# B&R Automation Studio project ControlPLC_DataDistribution (part 3)

#### Cyclic.sfc
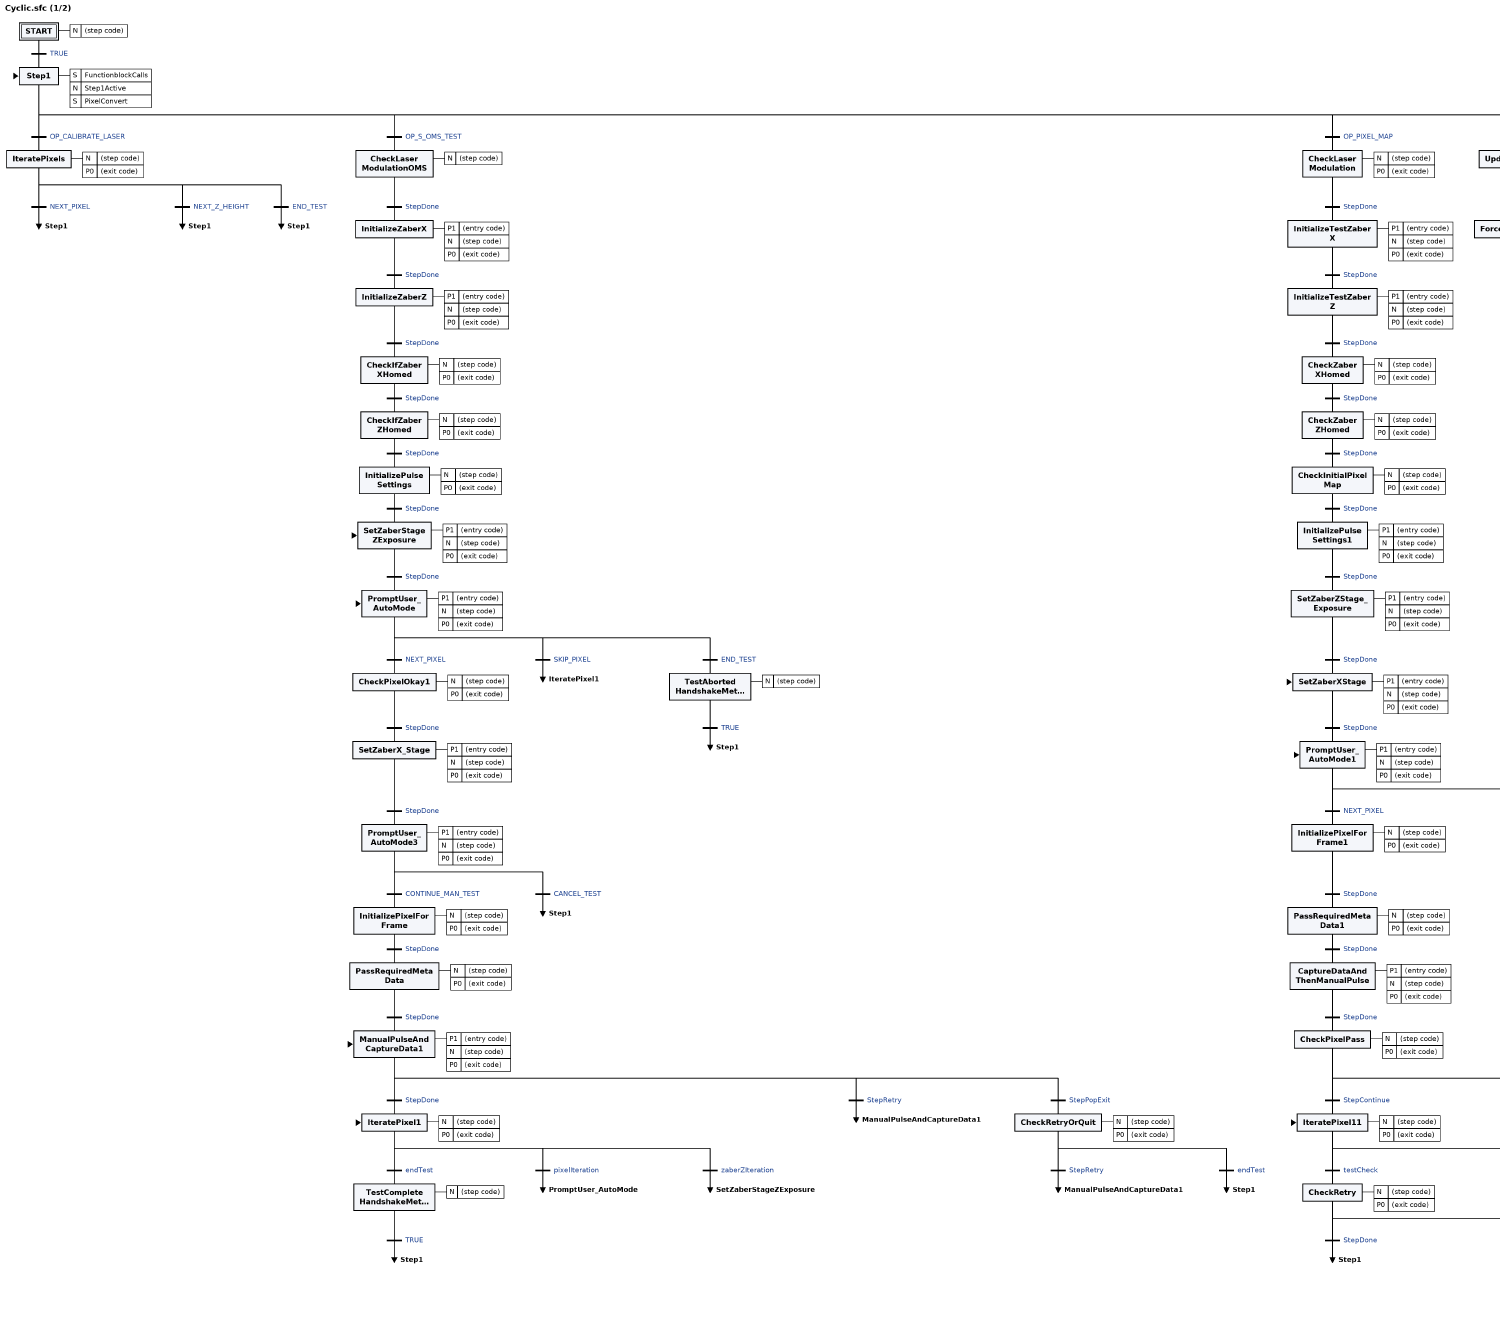
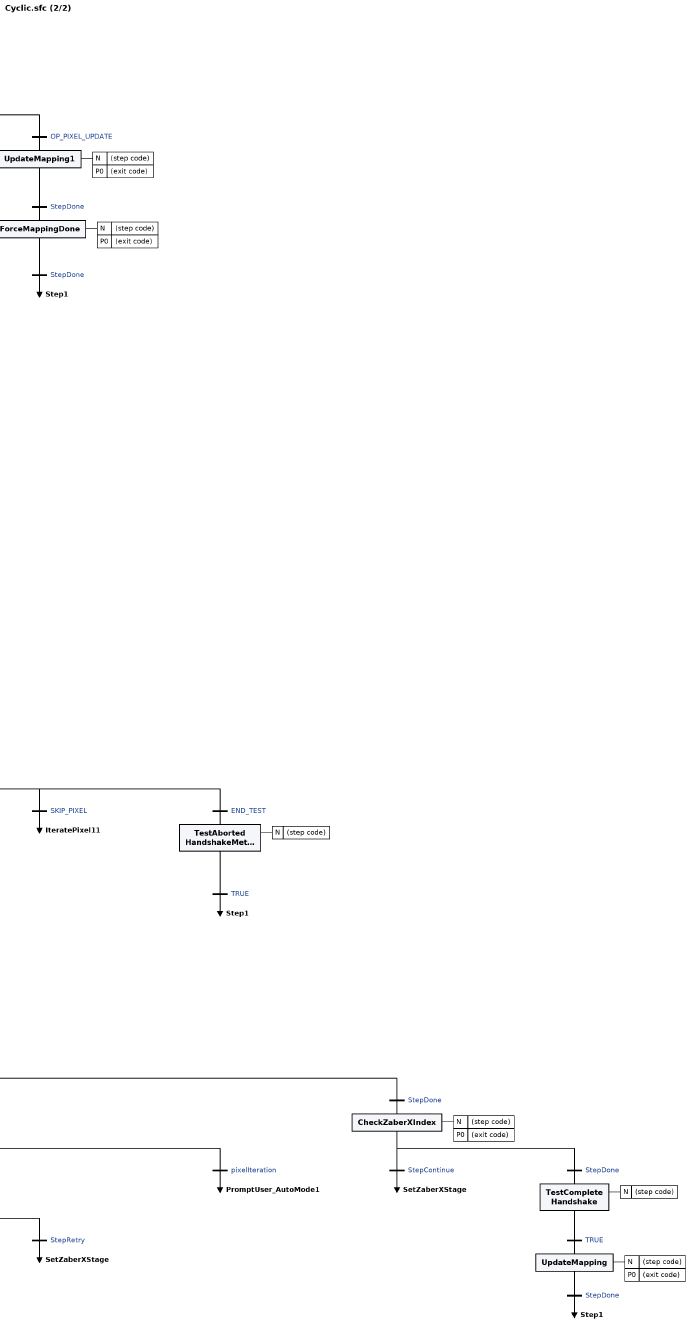
```iecst
PROGRAM _CYCLIC
INITIAL_STEP START:

SFCReset := FALSE;
END_STEP
TRANSITION FROM START TO Step1:=
TRUE
END_TRANSITION
IEC_STEP Step1:
FunctionblockCalls(S);
Step1Active(N);
PixelConvert(S);
END_STEP
TRANSITION FROM Step1 TO IteratePixels:=
OP_CALIBRATE_LASER
END_TRANSITION
TRANSITION FROM Step1 TO CheckLaserModulationOMS:=
OP_S_OMS_TEST
END_TRANSITION
STEP CheckLaserModulationOMS:
OP_S_OMS_TEST := FALSE;
task.internal.activeZaber2Index := 0;

StepDone := TRUE;
END_STEP
TRANSITION FROM CheckLaserModulationOMS TO InitializeZaberX:=
StepDone
END_TRANSITION
STEP InitializeZaberX:
OP_CALIBRATE_LASER := FALSE;
// initialize test
// init meta writer; Zome Zaber

Command.Command := gVFLCR.command.initializeOmsTestZaber1;

Command.Execute := TRUE;
Command();

IF Command.Done THEN
	StepDone := TRUE;
	Command.Execute := FALSE;
	Command();

ELSE
	StepDone := FALSE;
END_IF
END_STEP
ENTRY_ACTION
task.internal.activeZaber2Index := 0;
END_ACTION
EXIT_ACTION
StepDone := FALSE;
(* TODO: Insert Program *)
END_ACTION
TRANSITION FROM InitializeZaberX TO InitializeZaberZ:=
StepDone
END_TRANSITION
STEP InitializeZaberZ:
OP_CALIBRATE_LASER := FALSE;
// initialize test
// init meta writer; Zome Zaber

Command.Command := gVFLCR.command.initializeOmsTestZaber2;

Command.Execute := TRUE;
Command();

IF Command.Done THEN
	StepDone := TRUE;
	Command.Execute := FALSE;
	Command();

ELSE
	StepDone := FALSE;
END_IF
END_STEP
ENTRY_ACTION
task.internal.activeZaber2Index := 0;
END_ACTION
EXIT_ACTION
StepDone := FALSE;
(* TODO: Insert Program *)
END_ACTION
TRANSITION FROM InitializeZaberZ TO CheckIfZaberXHomed:=
StepDone
END_TRANSITION
STEP CheckIfZaberXHomed:
Command.Command := gVFLCR.command.checkZaber1Homed;

Command.Execute := TRUE;
Command();

IF Command.Done THEN
	StepDone := TRUE;
	Command.Execute := FALSE;
	Command();
ELSE
	StepDone := FALSE;
END_IF
END_STEP
EXIT_ACTION
StepDone := FALSE;
(* TODO: Insert Program *)
END_ACTION
TRANSITION FROM CheckIfZaberXHomed TO CheckIfZaberZHomed:=
StepDone
END_TRANSITION
STEP CheckIfZaberZHomed:
Command.Command := gVFLCR.command.checkZaber2Homed;

Command.Execute := TRUE;
Command();

IF Command.Done THEN
	StepDone := TRUE;
	Command.Execute := FALSE;
	Command();
ELSE
	StepDone := FALSE;
END_IF
END_STEP
EXIT_ACTION
StepDone := FALSE;
(* TODO: Insert Program *)
END_ACTION
TRANSITION FROM CheckIfZaberZHomed TO InitializePulseSettings:=
StepDone
END_TRANSITION
STEP InitializePulseSettings:
// initialize app with manual pulse pars; Will create directories for calibration test as well- Should be ok; Assuming data backup of last test to Nas is done by then
Command.Command := gVFLCR.command.initializeCalibration;

Command.pParameters := ADR(gManualPulseTypeSelected);
Command.sParameters := SIZEOF(gManualPulseTypeSelected);

Command.Execute := TRUE;
Command();

IF Command.Done THEN
	StepDone := TRUE;
	Command.Execute := FALSE;
	Command();
ELSE

	StepDone := FALSE;

END_IF
END_STEP
EXIT_ACTION
StepDone := FALSE;
(* TODO: Insert Program *)
END_ACTION
TRANSITION FROM InitializePulseSettings TO SetZaberStageZExposure:=
StepDone
END_TRANSITION
STEP SetZaberStageZExposure:

// Set Zaber height and camera exposure
Command.Command := gVFLCR.command.setZaber2PosAndExposure;

Command.pParameters := ADR(task.internal.adjustZaber2AndCamera);
Command.sParameters := SIZEOF(task.internal.adjustZaber2AndCamera);

Command.Execute := TRUE;
Command();

IF Command.Done THEN
	StepDone := TRUE;
	Command.Execute := FALSE;
	Command();
ELSE

	StepDone := FALSE;

END_IF
END_STEP
ENTRY_ACTION
task.internal.activePixelIndex := 0;

brsmemset( ADR(task.internal.adjustZaber2AndCamera), 0, SIZEOF(task.internal.adjustZaber2AndCamera) );

task.internal.adjustZaber2AndCamera.ZaberAbsolutePos_mm := Configuration.zaber2HeightArray[task.internal.activeZaber2Index];
task.internal.adjustZaber2AndCamera.ZaberMoveAbsolute := TRUE ;
task.internal.adjustZaber2AndCamera.CameraExposure := Configuration.zaber2HeightCameraExpoArray[task.internal.activeZaber2Index];
END_ACTION
EXIT_ACTION
StepDone := FALSE;
END_ACTION
TRANSITION FROM SetZaberStageZExposure TO PromptUser_AutoMode:=
StepDone
END_TRANSITION
STEP PromptUser_AutoMode:

IF NOT autoMode THEN

	task.internal.showPopUp := TRUE;
	task.internal.showNextPixel := TRUE;
	task.internal.showSkipPixel:= TRUE;

	IF task.internal.showPopUp THEN

		IF task.internal.activePixelIndex >= MACHINE_NUM_LASERS_TOTAL THEN

			task.internal.showNextPixel := FALSE;
			task.internal.showSkipPixel:= FALSE;

		ELSIF gVFLCR.status.vfpMap[task.internal.activePixelIndex , 1] = FALSE THEN

			// pixel is disabled
			//task.internal.msgId := TRUE;
			task.internal.showNextPixel := FALSE;

		ELSE

			// pixel is enabled
			//task.internal.msgId := TRUE;
			task.internal.showSkipPixel:= FALSE;

		END_IF

	END_IF

	IF task.internal.showPopUp <> 0 THEN

	END_IF

	//	IF messageHandler.cancel THEN
	//		messageHandler.cancel := 0;
	//		task.internal.msgId := FALSE;
	//		SFCReset := TRUE;
	//		gMachine.IN.CMD.Stop:= TRUE;
	//	END_IF

	//Once a selection is made we are good
	IF NEXT_PIXEL OR SKIP_PIXEL OR END_TEST THEN

		task.internal.showPopUp := FALSE;
		task.internal.showSkipPixel:= FALSE;
		task.internal.showNextPixel := FALSE;

	END_IF
ELSE
	IF gVFLCR.status.vfpMap[task.internal.activePixelIndex, 1] = FALSE THEN
		SKIP_PIXEL := TRUE;
	ELSE
		NEXT_PIXEL := TRUE;
	END_IF
END_IF
END_STEP
ENTRY_ACTION
task.internal.showPopUp := 0;
NEXT_PIXEL := FALSE;
SKIP_PIXEL := FALSE;
END_TEST := FALSE;

END_ACTION
EXIT_ACTION
NEXT_PIXEL := FALSE;
SKIP_PIXEL := FALSE;
END_TEST := FALSE;
END_ACTION
TRANSITION FROM PromptUser_AutoMode TO CheckPixelOkay1:=
NEXT_PIXEL
END_TRANSITION
TRANSITION FROM PromptUser_AutoMode TO IteratePixel1:=
SKIP_PIXEL
END_TRANSITION
(* @SFCISJUMP := 'IteratePixel1' *)
TRANSITION FROM PromptUser_AutoMode TO TestAbortedHandshakeMetaWriter:=
END_TEST
END_TRANSITION
STEP TestAbortedHandshakeMetaWriter:
Command.Command := gVFLCR.command.passAbortedHandshake;

Command.Execute := TRUE;
Command();

IF Command.Done THEN
	StepDone := TRUE;
	Command.Execute := FALSE;
	Command();
ELSE
	StepDone := FALSE;
END_IF
END_STEP
TRANSITION FROM TestAbortedHandshakeMetaWriter TO Step1:=
TRUE
END_TRANSITION
(* @SFCISJUMP := 'Step1' *)
STEP CheckPixelOkay1:
Command.Command := gVFLCR.command.checkMotionOk;
Command.Execute := TRUE;
Command();

IF Command.Done THEN
	StepDone := TRUE;
	Command.Execute := FALSE;
	Command();
ELSE
	StepDone := FALSE;
END_IF

END_STEP
EXIT_ACTION
StepDone := FALSE;
END_ACTION
TRANSITION FROM CheckPixelOkay1 TO SetZaberX_Stage:=
StepDone
END_TRANSITION
STEP SetZaberX_Stage:

// Set Zaber height and camera exposure
Command.Command := gVFLCR.command.setZaber1Pos;

Command.pParameters := ADR(task.internal.adjustZaber1);
Command.sParameters := SIZEOF(task.internal.adjustZaber1);

Command.Execute := TRUE;
Command();

IF Command.Done THEN
	StepDone := TRUE;
	Command.Execute := FALSE;
	Command();
ELSE

	StepDone := FALSE;

END_IF
END_STEP
ENTRY_ACTION

brsmemset( ADR(task.internal.adjustZaber1), 0, SIZEOF(task.internal.adjustZaber1) );

task.internal.adjustZaber1.ZaberAbsolutePos_mm := Configuration.zaber1Position + ((task.internal.activePixelIndex+1) * OPTICS_BOX_PIXEL_XY_OFFSET) ;
task.internal.adjustZaber1.ZaberMoveAbsolute := TRUE ;

END_ACTION
EXIT_ACTION
StepDone := FALSE;
END_ACTION
TRANSITION FROM SetZaberX_Stage TO PromptUser_AutoMode3:=
StepDone
END_TRANSITION
STEP PromptUser_AutoMode3:

IF NOT autoMode THEN

	task.internal.pausePopUp := TRUE;
	task.internal.continuePopUp := TRUE;
	task.internal.cancelPopUp := TRUE;

	IF task.internal.pausePopUp <> 0 THEN

	END_IF

	//Once a selection is made we are good
	IF CONTINUE_MAN_TEST OR CANCEL_TEST THEN

		task.internal.pausePopUp := FALSE;
		task.internal.continuePopUp:= FALSE;
		task.internal.cancelPopUp := FALSE;

	END_IF
ELSE
	CONTINUE_MAN_TEST := TRUE;
	task.internal.pausePopUp := FALSE;
	task.internal.continuePopUp:= FALSE;
	task.internal.cancelPopUp := FALSE;
END_IF
END_STEP
ENTRY_ACTION
task.internal.pausePopUp := 0;
CONTINUE_MAN_TEST := FALSE;
CANCEL_TEST := FALSE;

END_ACTION
EXIT_ACTION
CONTINUE_MAN_TEST := FALSE;
CANCEL_TEST := FALSE;
END_ACTION
TRANSITION FROM PromptUser_AutoMode3 TO InitializePixelForFrame:=
CONTINUE_MAN_TEST
END_TRANSITION
TRANSITION FROM PromptUser_AutoMode3 TO Step1:=
CANCEL_TEST
END_TRANSITION
(* @SFCISJUMP := 'Step1' *)
STEP InitializePixelForFrame:
Command.Command := gVFLCR.command.initializePixelForFrame;

task.internal.initializePixelParameters.activePixelIndex := task.internal.activePixelIndex;

Command.pParameters := ADR(task.internal.initializePixelParameters);
Command.sParameters := SIZEOF(task.internal.initializePixelParameters);

Command.Execute := TRUE;
Command();

IF Command.Done THEN
	StepDone := TRUE;
	Command.Execute := FALSE;
	Command();
ELSE

	StepDone := FALSE;

END_IF
END_STEP
EXIT_ACTION
StepDone := FALSE;
END_ACTION
TRANSITION FROM InitializePixelForFrame TO PassRequiredMetaData:=
StepDone
END_TRANSITION
STEP PassRequiredMetaData:
Command.Command := gVFLCR.command.passRequiredMetaData;

Command.Execute := TRUE;
Command();

IF Command.Done THEN
	StepDone := TRUE;
	Command.Execute := FALSE;
	Command();
ELSE
	StepDone := FALSE;
END_IF
END_STEP
EXIT_ACTION
StepDone := FALSE;
END_ACTION
TRANSITION FROM PassRequiredMetaData TO ManualPulseAndCaptureData1:=
StepDone
END_TRANSITION
STEP ManualPulseAndCaptureData1:
Command.Command := gVFLCR.command.manualPulse;

Command.pParameters := ADR(task.internal.manualPulse);
Command.sParameters := SIZEOF(task.internal.manualPulse);

Command.Execute := TRUE;
Command();

IF Command.Done THEN
	StepDone := TRUE;
	task.internal.failedImageCaptureRetry := 0;
	Command.Execute := FALSE;
	Command();
ELSIF Command.Error THEN
	IF task.internal.failedImageCaptureRetry < task.internal.numOfRetries THEN
		StepRetry := TRUE;
		task.internal.failedImageCaptureRetry := task.internal.failedImageCaptureRetry +1;
		Command.Execute := FALSE;
		Command();
	ELSE
		task.internal.failedImageCaptureRetry := 0;
		StepDone := FALSE;
		StepRetry := FALSE;
		StepPopExit := TRUE;
		Command.Execute := FALSE;
		Command();
	END_IF
ELSE
	StepDone := FALSE;
END_IF
END_STEP
ENTRY_ACTION
task.internal.numOfRetries := 4;
END_ACTION
EXIT_ACTION
StepRetry := FALSE;
StepDone := FALSE;
StepPopExit := FALSE;
END_ACTION
TRANSITION FROM ManualPulseAndCaptureData1 TO IteratePixel1:=
StepDone
END_TRANSITION
TRANSITION FROM ManualPulseAndCaptureData1 TO ManualPulseAndCaptureData1:=
StepRetry
END_TRANSITION
(* @SFCISJUMP := 'ManualPulseAndCaptureData1' *)
TRANSITION FROM ManualPulseAndCaptureData1 TO CheckRetryOrQuit:=
StepPopExit
END_TRANSITION
STEP CheckRetryOrQuit:
task.internal.showErrorMessage := TRUE;

IF task.internal.showErrorMessage <> 0 THEN

END_IF

IF CLOSE_POPUP  THEN

	task.internal.showErrorMessage := FALSE;
	endTest :=TRUE;
	StepRetry:=FALSE;

END_IF

IF RETRY_POPUP  THEN

	task.internal.showErrorMessage := FALSE;
	StepRetry:=TRUE;
	endTest :=FALSE;

END_IF
END_STEP
EXIT_ACTION
endTest := FALSE;
StepRetry := FALSE;
END_ACTION
TRANSITION FROM CheckRetryOrQuit TO ManualPulseAndCaptureData1:=
StepRetry
END_TRANSITION
(* @SFCISJUMP := 'ManualPulseAndCaptureData1' *)
TRANSITION FROM CheckRetryOrQuit TO Step1:=
endTest
END_TRANSITION
(* @SFCISJUMP := 'Step1' *)
STEP IteratePixel1:
task.internal.activePixelIndex := task.internal.activePixelIndex + 1;

IF task.internal.activePixelIndex >= MACHINE_NUM_LASERS_TOTAL THEN
	IF  task.internal.activeZaber2Index < 10 THEN // 0-10 point reading with 5 being zero offset position and 5 reading on either side
		zaberZIteration := TRUE;
		task.internal.activeZaber2Index := task.internal.activeZaber2Index + 1;
	ELSE
		endTest := TRUE;
	END_IF
ELSE
	pixelIteration := TRUE;
END_IF
END_STEP
EXIT_ACTION

pixelIteration := FALSE;
zaberZIteration := FALSE;
endTest := FALSE;
END_ACTION
TRANSITION FROM IteratePixel1 TO TestCompleteHandshakeMetaWriter:=
endTest
END_TRANSITION
TRANSITION FROM IteratePixel1 TO PromptUser_AutoMode:=
pixelIteration
END_TRANSITION
(* @SFCISJUMP := 'PromptUser_AutoMode' *)
TRANSITION FROM IteratePixel1 TO SetZaberStageZExposure:=
zaberZIteration
END_TRANSITION
(* @SFCISJUMP := 'SetZaberStageZExposure' *)
STEP TestCompleteHandshakeMetaWriter:
endTest := FALSE;

Command.Command := gVFLCR.command.passCompleteHandshake;

Command.Execute := TRUE;
Command();

IF Command.Done THEN
	StepDone := TRUE;
	omsTestComplete := TRUE;
	Command.Execute := FALSE;
	Command();
ELSE
	StepDone := FALSE;
END_IF
END_STEP
TRANSITION FROM TestCompleteHandshakeMetaWriter TO Step1:=
TRUE
END_TRANSITION
(* @SFCISJUMP := 'Step1' *)
TRANSITION FROM Step1 TO CheckLaserModulation:=
OP_PIXEL_MAP
END_TRANSITION
STEP CheckLaserModulation:
OP_PIXEL_MAP := FALSE;
omsTestComplete := FALSE;
endTest := FALSE;
pixelIteration := FALSE;

FOR loopVar := 0 TO MACHINE_MAI_LASERS_TOTAL BY 1 DO
	pixelIgnoreList[loopVar] := FALSE;
END_FOR

StepDone := TRUE;

END_STEP
EXIT_ACTION
StepDone := FALSE;
END_ACTION
TRANSITION FROM CheckLaserModulation TO InitializeTestZaberX:=
StepDone
END_TRANSITION
STEP InitializeTestZaberX:
OP_CALIBRATE_LASER := FALSE;
// initialize test
// init meta writer; Zome Zaber

Command.Command := gVFLCR.command.initializeOmsTestZaber1;

Command.Execute := TRUE;
Command();

IF Command.Done THEN
	StepDone := TRUE;
	Command.Execute := FALSE;
	Command();

ELSE
	StepDone := FALSE;
END_IF
END_STEP
ENTRY_ACTION
task.internal.activeZaber2Index := 0;
END_ACTION
EXIT_ACTION
StepDone := FALSE;
END_ACTION
TRANSITION FROM InitializeTestZaberX TO InitializeTestZaberZ:=
StepDone
END_TRANSITION
STEP InitializeTestZaberZ:
OP_CALIBRATE_LASER := FALSE;
// initialize test
// init meta writer; Zome Zaber

Command.Command := gVFLCR.command.initializeOmsTestZaber2;

Command.Execute := TRUE;
Command();

IF Command.Done THEN
	StepDone := TRUE;
	Command.Execute := FALSE;
	Command();

ELSE
	StepDone := FALSE;
END_IF
END_STEP
ENTRY_ACTION
task.internal.activeZaber2Index := 0;
END_ACTION
EXIT_ACTION
StepDone := FALSE;
END_ACTION
TRANSITION FROM InitializeTestZaberZ TO CheckZaberXHomed:=
StepDone
END_TRANSITION
STEP CheckZaberXHomed:
Command.Command := gVFLCR.command.checkZaber1Homed;

Command.Execute := TRUE;
Command();

IF Command.Done THEN
	StepDone := TRUE;
	Command.Execute := FALSE;
	Command();
ELSE
	StepDone := FALSE;
END_IF
END_STEP
EXIT_ACTION
StepDone := FALSE;
END_ACTION
TRANSITION FROM CheckZaberXHomed TO CheckZaberZHomed:=
StepDone
END_TRANSITION
STEP CheckZaberZHomed:
Command.Command := gVFLCR.command.checkZaber2Homed;

Command.Execute := TRUE;
Command();

IF Command.Done THEN
	StepDone := TRUE;
	Command.Execute := FALSE;
	Command();
ELSE
	StepDone := FALSE;
END_IF
END_STEP
EXIT_ACTION
StepDone := FALSE;
END_ACTION
TRANSITION FROM CheckZaberZHomed TO CheckInitialPixelMap:=
StepDone
END_TRANSITION
STEP CheckInitialPixelMap:
task.status.allPixelsMapped := stateAllTrue(gVFLCR.status.pixelMapped, FALSE);

FOR task.internal.rackNumber := 0 TO MACHINE_MAI_LASER_RACKS  DO
	FOR task.internal.laserNumber := 0 TO MACHINE_MAI_LASERS_PER_RACK  DO
		gVFLCR.status.vfpMap[task.internal.laserNumber,task.internal.rackNumber] := TRUE;
		//task.internal.laserNumber := task.internal.laserNumber +1;
	END_FOR
	//task.internal.rackNumber := task.internal.rackNumber +1;
END_FOR

IF task.status.allPixelsMapped THEN
	StepDone := TRUE;
ELSE
	StepDone := FALSE;

	Command.Command := gVFLCR.command.laserRackRemap;

	Command.Execute := TRUE;
	Command();

	IF Command.Done THEN
		StepDone := TRUE;
		Command.Execute := FALSE;
		Command();
	ELSIF Command.Error THEN
		StepError := TRUE;
	END_IF

END_IF
END_STEP
EXIT_ACTION
StepDone := FALSE;
END_ACTION
TRANSITION FROM CheckInitialPixelMap TO InitializePulseSettings1:=
StepDone
END_TRANSITION
STEP InitializePulseSettings1:
// initialize app with manual pulse pars; Will create directories for calibration test as well- Should be ok; Assuming data backup of last test to Nas is done by then
Command.Command := gVFLCR.command.initializeCalibration;

Command.pParameters := ADR(gManualPulseTypeSelected);
Command.sParameters := SIZEOF(gManualPulseTypeSelected);

Command.Execute := TRUE;
Command();

IF Command.Done THEN
	StepDone := TRUE;
	Command.Execute := FALSE;
	Command();
ELSE

	StepDone := FALSE;

END_IF
END_STEP
ENTRY_ACTION
brsmemset(ADR(derivedMappingList), 0, SIZEOF(derivedMappingList));
END_ACTION
EXIT_ACTION
StepDone := FALSE;
END_ACTION
TRANSITION FROM InitializePulseSettings1 TO SetZaberZStage_Exposure:=
StepDone
END_TRANSITION
STEP SetZaberZStage_Exposure:

task.internal.adjustZaber1.ZaberAbsolutePos_mm := Configuration.zaber1Position;
// Set Zaber height and camera exposure
Command.Command := gVFLCR.command.setZaber2PosAndExposure;

Command.pParameters := ADR(task.internal.adjustZaber2AndCamera);
Command.sParameters := SIZEOF(task.internal.adjustZaber2AndCamera);

Command.Execute := TRUE;
Command();

IF Command.Done THEN
	StepDone := TRUE;
	Command.Execute := FALSE;
	Command();
ELSE

	StepDone := FALSE;

END_IF
END_STEP
ENTRY_ACTION

task.internal.actualPixelMapIndex :=0; // used for derived mapping list
task.internal.activeZaber1Index := 0; // Initialized once at the start of the test
task.internal.failedImageCaptureRetry := 0; // Reset Retry count

brsmemset( ADR(task.internal.adjustZaber2AndCamera), 0, SIZEOF(task.internal.adjustZaber2AndCamera) );

task.internal.adjustZaber2AndCamera.ZaberAbsolutePos_mm := Configuration.zaber2HeightArray[5]; // only use middle height
task.internal.adjustZaber2AndCamera.ZaberMoveAbsolute := TRUE ;
task.internal.adjustZaber2AndCamera.CameraExposure := Configuration.zaber2HeightCameraExpoArray[5];
END_ACTION
EXIT_ACTION
StepDone := FALSE;
END_ACTION
TRANSITION FROM SetZaberZStage_Exposure TO SetZaberXStage:=
StepDone
END_TRANSITION
STEP SetZaberXStage:

// Set Zaber height and camera exposure
Command.Command := gVFLCR.command.setZaber1Pos;

FOR loopVar := 0 TO MACHINE_MAI_LASERS_TOTAL BY 1 DO
	IF pixelIgnoreList[task.internal.activePixelIndex] = TRUE THEN
		task.internal.activePixelIndex := task.internal.activePixelIndex + 1;
	ELSE
		EXIT;
	END_IF
END_FOR

Command.pParameters := ADR(task.internal.adjustZaber1);
Command.sParameters := SIZEOF(task.internal.adjustZaber1);

Command.Execute := TRUE;
Command();

IF Command.Done THEN
	StepDone := TRUE;
	Command.Execute := FALSE;
	Command();
ELSE

	StepDone := FALSE;

END_IF
END_STEP
ENTRY_ACTION
task.internal.activePixelIndex := 0; // used to iterate through all pixels during pixel mapping

FOR loopVar := 0 TO MACHINE_MAI_LASERS_TOTAL BY 1 DO
	IF pixelIgnoreList[task.internal.activePixelIndex] = TRUE THEN
		task.internal.activePixelIndex := task.internal.activePixelIndex + 1;
	ELSE
		EXIT;
	END_IF
END_FOR

brsmemset( ADR(task.internal.adjustZaber1), 0, SIZEOF(task.internal.adjustZaber1) );

task.internal.adjustZaber1.ZaberAbsolutePos_mm := Configuration.zaber1Position + ((task.internal.activeZaber1Index+1) * OPTICS_BOX_PIXEL_XY_OFFSET) ;
task.internal.adjustZaber1.ZaberMoveAbsolute := TRUE ;

END_ACTION
EXIT_ACTION
StepDone := FALSE;
END_ACTION
TRANSITION FROM SetZaberXStage TO PromptUser_AutoMode1:=
StepDone
END_TRANSITION
STEP PromptUser_AutoMode1:

IF NOT autoMode THEN
	task.internal.showPopUp := TRUE;
	task.internal.showNextPixel := TRUE;
	task.internal.showSkipPixel:= TRUE;

	IF task.internal.showPopUp THEN

		IF task.internal.activePixelIndex >= MACHINE_NUM_LASERS_TOTAL THEN

			task.internal.showNextPixel := FALSE;
			task.internal.showSkipPixel:= FALSE;

		ELSIF pixelIgnoreList[task.internal.activePixelIndex] = TRUE THEN

			// pixel is disabled
			//task.internal.msgId := TRUE;
			task.internal.showNextPixel := FALSE;

		ELSE

			// pixel is enabled
			//task.internal.msgId := TRUE;
			task.internal.showSkipPixel:= FALSE;

		END_IF

	END_IF

	IF task.internal.showPopUp <> 0 THEN

	END_IF

	//	IF messageHandler.cancel THEN
	//		messageHandler.cancel := 0;
	//		task.internal.msgId := FALSE;
	//		SFCReset := TRUE;
	//		gMachine.IN.CMD.Stop:= TRUE;
	//	END_IF

	//Once a selection is made we are good
	IF NEXT_PIXEL OR SKIP_PIXEL OR END_TEST THEN

		task.internal.showPopUp := FALSE;
		task.internal.showSkipPixel:= FALSE;
		task.internal.showNextPixel := FALSE;

	END_IF
ELSE
	IF pixelIgnoreList[task.internal.activePixelIndex] = TRUE THEN
		SKIP_PIXEL := TRUE;
	ELSE
		NEXT_PIXEL := TRUE;
	END_IF
END_IF
END_STEP
ENTRY_ACTION
task.internal.showPopUp := 0;
NEXT_PIXEL := FALSE;
SKIP_PIXEL := FALSE;
END_TEST := FALSE;
END_ACTION
EXIT_ACTION
NEXT_PIXEL := FALSE;
SKIP_PIXEL := FALSE;
END_TEST := FALSE;
END_ACTION
TRANSITION FROM PromptUser_AutoMode1 TO InitializePixelForFrame1:=
NEXT_PIXEL
END_TRANSITION
TRANSITION FROM PromptUser_AutoMode1 TO IteratePixel11:=
SKIP_PIXEL
END_TRANSITION
(* @SFCISJUMP := 'IteratePixel11' *)
TRANSITION FROM PromptUser_AutoMode1 TO TestAbortedHandshakeMetaWriter1:=
END_TEST
END_TRANSITION
STEP TestAbortedHandshakeMetaWriter1:
Command.Command := gVFLCR.command.passAbortedHandshake;

Command.Execute := TRUE;
Command();

IF Command.Done THEN
	StepDone := TRUE;
	Command.Execute := FALSE;
	Command();
ELSE
	StepDone := FALSE;
END_IF
END_STEP
TRANSITION FROM TestAbortedHandshakeMetaWriter1 TO Step1:=
TRUE
END_TRANSITION
(* @SFCISJUMP := 'Step1' *)
STEP InitializePixelForFrame1:
Command.Command := gVFLCR.command.initializePixelForFrame;

task.internal.initializePixelParameters.activePixelIndex := task.internal.activePixelIndex;

Command.pParameters := ADR(task.internal.initializePixelParameters);
Command.sParameters := SIZEOF(task.internal.initializePixelParameters);

Command.Execute := TRUE;
Command();

IF Command.Done THEN
	StepDone := TRUE;
	Command.Execute := FALSE;
	Command();
ELSE

	StepDone := FALSE;

END_IF
END_STEP
EXIT_ACTION
StepDone := FALSE;
END_ACTION
TRANSITION FROM InitializePixelForFrame1 TO PassRequiredMetaData1:=
StepDone
END_TRANSITION
STEP PassRequiredMetaData1:
Command.Command := gVFLCR.command.passRequiredMetaData;

Command.Execute := TRUE;
Command();

IF Command.Done THEN
	StepDone := TRUE;
	Command.Execute := FALSE;
	Command();
ELSE
	StepDone := FALSE;
END_IF
END_STEP
EXIT_ACTION
StepDone := FALSE;
END_ACTION
TRANSITION FROM PassRequiredMetaData1 TO CaptureDataAndThenManualPulse:=
StepDone
END_TRANSITION
STEP CaptureDataAndThenManualPulse:
Command.Command := gVFLCR.command.manualPulse;

Command.pParameters := ADR(task.internal.manualPulse);
Command.sParameters := SIZEOF(task.internal.manualPulse);

Command.Execute := TRUE;
Command();

IF Command.Done THEN
	StepDone := TRUE;
	Command.Execute := FALSE;
	Command();
ELSIF Command.Error THEN
	StepDone := TRUE;
	Command.Execute := FALSE;
	Command();

END_IF
END_STEP
ENTRY_ACTION
task.internal.numOfRetries := 3;
END_ACTION
EXIT_ACTION
StepDone := FALSE;
END_ACTION
TRANSITION FROM CaptureDataAndThenManualPulse TO CheckPixelPass:=
StepDone
END_TRANSITION
STEP CheckPixelPass:
task.internal.rackNumber := 0;
task.internal.laserNumber :=0;

IF gVFLCR.status.frameCaptured THEN
	//task.internal.actualPixelMapIndex := task.internal.actualPixelMapIndex +1;
	FOR task.internal.rackNumber := 0 TO MACHINE_MAI_LASER_RACKS  DO
		IF NOT (gVFLCR.status.vfpMap[task.internal.activePixelIndex, 1] = FALSE) THEN
			FOR task.internal.laserNumber := 0 TO MACHINE_MAI_LASERS_PER_RACK  DO
				IF gmapRackLaser_to_Pixel[task.internal.rackNumber,task.internal.laserNumber] = task.internal.activePixelIndex THEN
					derivedMappingList[task.internal.rackNumber,task.internal.laserNumber] := task.internal.activeZaber1Index;
					pixelIgnoreList[task.internal.activePixelIndex] := TRUE;
					gVFLCR.status.frameCaptured := FALSE;
				END_IF
			END_FOR
		END_IF
	END_FOR
			StepDone := TRUE;
			StepContinue := FALSE;

		ELSE
			StepDone := FALSE;
			StepContinue := TRUE;
		END_IF

END_STEP
EXIT_ACTION
StepDone := FALSE;
StepContinue := FALSE;
END_ACTION
TRANSITION FROM CheckPixelPass TO IteratePixel11:=
StepContinue
END_TRANSITION
TRANSITION FROM CheckPixelPass TO CheckZaberXIndex:=
StepDone
END_TRANSITION
STEP CheckZaberXIndex:
IF task.internal.activeZaber1Index < (MACHINE_NUM_LASERS_TOTAL - 1) THEN
	StepContinue := TRUE;
	task.internal.activeZaber1Index:= task.internal.activeZaber1Index +1 ;
ELSE
	StepDone := TRUE;
END_IF

END_STEP
EXIT_ACTION
StepDone := FALSE;
StepContinue := FALSE;
END_ACTION
TRANSITION FROM CheckZaberXIndex TO SetZaberXStage:=
StepContinue
END_TRANSITION
(* @SFCISJUMP := 'SetZaberXStage' *)
TRANSITION FROM CheckZaberXIndex TO TestCompleteHandshake:=
StepDone
END_TRANSITION
STEP TestCompleteHandshake:
endTest := FALSE;

Command.Command := gVFLCR.command.passCompleteHandshake;

Command.Execute := TRUE;
Command();

IF Command.Done THEN
	StepDone := TRUE;
	omsTestComplete := TRUE;
	Command.Execute := FALSE;
	Command();
ELSE
	StepDone := FALSE;
END_IF
END_STEP
TRANSITION FROM TestCompleteHandshake TO UpdateMapping:=
TRUE
END_TRANSITION
STEP UpdateMapping:

FOR task.internal.rackIndex := 0 TO (MACHINE_NUM_LASER_RACKS-1)  DO
	FOR task.internal.laserIndex := 0 TO (MACHINE_NUM_LASERS_PER_RACK-1) DO

		IF gVFLCR.status.vfpMap[gmapRackLaser_to_Pixel[task.internal.rackIndex,task.internal.laserIndex],1 ] = TRUE
			AND (((task.internal.rackIndex*MACHINE_NUM_LASERS_PER_RACK) + task.internal.laserIndex) < MACHINE_NUM_LASERS_TOTAL) THEN
			gmapRackLaser_to_Pixel[task.internal.rackIndex,task.internal.laserIndex] := derivedMappingList[task.internal.rackIndex,task.internal.laserIndex ];
			//task.internal.laserNumber := task.internal.laserNumber +1;
			gmapPixel_to_Rack[derivedMappingList[task.internal.rackIndex,task.internal.laserIndex]] := task.internal.rackIndex;
			gmapPixel_to_Laser[derivedMappingList[task.internal.rackIndex,task.internal.laserIndex]] := task.internal.laserIndex;
		END_IF
	END_FOR
END_FOR

FOR task.internal.clearListPixelNumber := 0 TO MACHINE_NUM_LASERS_TOTAL-1 DO
	pixelIgnoreList[task.internal.clearListPixelNumber] := FALSE;
END_FOR
StepDone := TRUE;
END_STEP
EXIT_ACTION
StepDone:=FALSE;
(* TODO: Insert Program *)
END_ACTION
TRANSITION FROM UpdateMapping TO Step1:=
StepDone
END_TRANSITION
(* @SFCISJUMP := 'Step1' *)
STEP IteratePixel11:
task.internal.activePixelIndex := task.internal.activePixelIndex + 1;

FOR loopVar := 0 TO MACHINE_MAI_LASERS_TOTAL BY 1 DO
	IF pixelIgnoreList[task.internal.activePixelIndex] = TRUE THEN
		task.internal.activePixelIndex := task.internal.activePixelIndex + 1;
	ELSE
		EXIT;
	END_IF
END_FOR

IF task.internal.activePixelIndex < MACHINE_NUM_LASERS_TOTAL  THEN

	pixelIteration := TRUE;
	testCheck := FALSE;

ELSE
	pixelIteration := FALSE;
	testCheck:= TRUE;
END_IF

END_STEP
EXIT_ACTION
pixelIteration := FALSE;
testError := FALSE;
END_ACTION
TRANSITION FROM IteratePixel11 TO CheckRetry:=
testCheck
END_TRANSITION
TRANSITION FROM IteratePixel11 TO PromptUser_AutoMode1:=
pixelIteration
END_TRANSITION
(* @SFCISJUMP := 'PromptUser_AutoMode1' *)
STEP CheckRetry:

task.internal.showErrorMessage := TRUE;

IF task.internal.showErrorMessage <> 0 THEN

END_IF

IF CLOSE_POPUP  THEN

	task.internal.showErrorMessage := FALSE;
	StepDone :=TRUE;
	StepRetry:=FALSE;

END_IF

IF RETRY_POPUP  THEN

	task.internal.showErrorMessage := FALSE;
	StepRetry:=TRUE;
	StepDone :=FALSE;

END_IF
END_STEP
EXIT_ACTION
pixelIteration := FALSE;
testError := FALSE;
StepDone := FALSE;
StepRetry:=FALSE;
END_ACTION
TRANSITION FROM CheckRetry TO Step1:=
StepDone
END_TRANSITION
(* @SFCISJUMP := 'Step1' *)
TRANSITION FROM CheckRetry TO SetZaberXStage:=
StepRetry
END_TRANSITION
(* @SFCISJUMP := 'SetZaberXStage' *)
TRANSITION FROM Step1 TO UpdateMapping1:=
OP_PIXEL_UPDATE
END_TRANSITION
STEP UpdateMapping1:

FOR task.internal.rackIndex := 0 TO (MACHINE_NUM_LASER_RACKS-1)  DO
	FOR task.internal.laserIndex := 0 TO (MACHINE_NUM_LASERS_PER_RACK-1) DO

		IF gVFLCR.status.vfpMap[gmapRackLaser_to_Pixel[task.internal.rackIndex,task.internal.laserIndex],1 ] = TRUE
			AND ((task.internal.rackIndex*(MACHINE_NUM_LASERS_PER_RACK) + task.internal.laserIndex) < MACHINE_NUM_LASERS_TOTAL) THEN
			gmapRackLaser_to_Pixel[task.internal.rackIndex,task.internal.laserIndex] := derivedMappingList[task.internal.rackIndex,task.internal.laserIndex ];
		//task.internal.laserNumber := task.internal.laserNumber +1;
			gmapPixel_to_Rack[derivedMappingList[task.internal.rackIndex,task.internal.laserIndex]] := task.internal.rackIndex;
			gmapPixel_to_Laser[derivedMappingList[task.internal.rackIndex,task.internal.laserIndex]] := task.internal.laserIndex;
		END_IF
	END_FOR
END_FOR

FOR task.internal.clearListPixelNumber := 0 TO (MACHINE_NUM_LASERS_TOTAL-1) DO
	pixelIgnoreList[task.internal.clearListPixelNumber] := FALSE;
END_FOR
StepDone := TRUE;

END_STEP
EXIT_ACTION
StepDone:=FALSE;
(* TODO: Insert Program *)
END_ACTION
TRANSITION FROM UpdateMapping1 TO ForceMappingDone:=
StepDone
END_TRANSITION
STEP ForceMappingDone:

Command.Command := gVFLCR.command.forceMappingDone;
Command.Execute := TRUE;
Command();

IF Command.Done THEN
	StepDone := TRUE;
	Command.Execute := FALSE;
	Command();
ELSE
	StepDone := FALSE;
END_IF

END_STEP
EXIT_ACTION
StepDone := FALSE;
END_ACTION
TRANSITION FROM ForceMappingDone TO Step1:=
StepDone
END_TRANSITION
(* @SFCISJUMP := 'Step1' *)
STEP IteratePixels:
task.internal.activePixelIndex := task.internal.activePixelIndex + 1;

IF task.internal.activePixelIndex >= 75 THEN
	IF task.internal.activeZaber2Index < 10 THEN
		// Next Z height
		NEXT_PIXEL := FALSE;
		END_TEST := FALSE;
		NEXT_Z_HEIGHT := TRUE;
	ELSE
		NEXT_PIXEL := FALSE;
		END_TEST := TRUE;
		NEXT_Z_HEIGHT := FALSE;
	END_IF
ELSE
	NEXT_PIXEL := TRUE;
	END_TEST := FALSE;
	NEXT_Z_HEIGHT := FALSE;
END_IF

END_STEP
EXIT_ACTION
NEXT_PIXEL := FALSE;
END_TEST := FALSE;
NEXT_Z_HEIGHT := FALSE;
END_ACTION
TRANSITION FROM IteratePixels TO Step1:=
NEXT_PIXEL
END_TRANSITION
(* @SFCISJUMP := 'Step1' *)
TRANSITION FROM IteratePixels TO Step1:=
NEXT_Z_HEIGHT
END_TRANSITION
(* @SFCISJUMP := 'Step1' *)
TRANSITION FROM IteratePixels TO Step1:=
END_TEST
END_TRANSITION
(* @SFCISJUMP := 'Step1' *)
END_PROGRAM
```

#### Init.st
```iecst
PROGRAM _INIT

	registerStateBool( gSFCControlApi.status.sOMSModeActive, 'SOMS mode active', task.internal.somsTestType );
	registerStateBool( gSFCControlApi.status.sOMSModeActive, 'Pixel Mapping Test active', task.internal.pixelMappingTestType );
	registerStateBool( gSFCControlApi.status.sOMSTestComplete, 'SOMS mode active', omsTestComplete );

END_PROGRAM
```

#### PixelConvert.st
```iecst
ACTION PixelConvert:

	IF (task.internal.activePixelIndex <= MACHINE_MAI_LASERS_TOTAL) THEN
		task.internal.manualPulse.Laser := gmapPixel_to_Laser[task.internal.activePixelIndex];
		task.internal.manualPulse.Rack := gmapPixel_to_Rack[task.internal.activePixelIndex];
	END_IF

	// Monitor test type set on HMI ======================================================================
	IF task.internal.pixelMappingTestType AND NOT task.internal._PixelMappingTestType THEN

		gManualPulseTypeSelected := VFLCR_TEST_TYPE_PIXEL_MAPPING;

		task.internal.calibrationTestType := FALSE;
		task.internal.dirtyVerificationTestType := FALSE;
		task.internal.cleanVerificationTestType := FALSE;
		task.internal.lowPowerTestType := FALSE;
		task.internal.somsTestType := FALSE;
		task.internal.highPowerTestType := FALSE;
	END_IF

	IF task.internal.calibrationTestType AND NOT task.internal._CalibrationTestType THEN

		gManualPulseTypeSelected := VFLCR_TEST_TYPE_CALIBRATION;

		task.internal.dirtyVerificationTestType := FALSE;
		task.internal.cleanVerificationTestType := FALSE;
		task.internal.lowPowerTestType := FALSE;
		task.internal.somsTestType := FALSE;
		task.internal.pixelMappingTestType := FALSE;
		task.internal.highPowerTestType := FALSE;
	END_IF

	IF task.internal.dirtyVerificationTestType AND NOT task.internal._DirtyVerificationTestType THEN

		gManualPulseTypeSelected := VFLCR_TEST_TYPE_VERIFY_DIRTY;

		task.internal.calibrationTestType := FALSE;
		task.internal.cleanVerificationTestType := FALSE;
		task.internal.lowPowerTestType := FALSE;
		task.internal.somsTestType := FALSE;
		task.internal.pixelMappingTestType := FALSE;
		task.internal.highPowerTestType := FALSE;
	END_IF

	IF task.internal.cleanVerificationTestType AND NOT task.internal._CleanVerificationTestType THEN

		gManualPulseTypeSelected := VFLCR_TEST_TYPE_VERIFY_CLEAN;

		task.internal.calibrationTestType := FALSE;
		task.internal.dirtyVerificationTestType := FALSE;
		task.internal.lowPowerTestType := FALSE;
		task.internal.somsTestType := FALSE;
		task.internal.pixelMappingTestType := FALSE;
	END_IF

	IF task.internal.lowPowerTestType AND NOT task.internal._LowPowerTestType THEN

		gManualPulseTypeSelected := VFLCR_TEST_TYPE_LOW_POWER_CHECK;

		task.internal.calibrationTestType := FALSE;
		task.internal.dirtyVerificationTestType := FALSE;
		task.internal.cleanVerificationTestType := FALSE;
		task.internal.somsTestType := FALSE;
		task.internal.pixelMappingTestType := FALSE;
		task.internal.highPowerTestType := FALSE;
	END_IF

	IF task.internal.somsTestType AND NOT task.internal._somsTestType THEN

		gManualPulseTypeSelected := VFLCR_TEST_TYPE_SOMS;

		task.internal.calibrationTestType := FALSE;
		task.internal.dirtyVerificationTestType := FALSE;
		task.internal.cleanVerificationTestType := FALSE;
		task.internal.lowPowerTestType := FALSE;
		task.internal.pixelMappingTestType := FALSE;
		task.internal.highPowerTestType := FALSE;
	END_IF

	IF task.internal.highPowerTestType AND NOT task.internal._HighPowerTestType THEN

		gManualPulseTypeSelected := VFLCR_TEST_TYPE_HIGH_POWER;

		task.internal.calibrationTestType := FALSE;
		task.internal.dirtyVerificationTestType := FALSE;
		task.internal.cleanVerificationTestType := FALSE;
		task.internal.somsTestType := FALSE;
		task.internal.lowPowerTestType := FALSE;
		task.internal.pixelMappingTestType := FALSE;
	END_IF

	task.internal._CalibrationTestType 			:= task.internal.calibrationTestType;
	task.internal._DirtyVerificationTestType 	:= task.internal.dirtyVerificationTestType;
	task.internal._CleanVerificationTestType 	:= task.internal.cleanVerificationTestType;
	task.internal._LowPowerTestType 			:= task.internal.lowPowerTestType;
	task.internal._somsTestType					:= task.internal.somsTestType;
	task.internal._PixelMappingTestType			:= task.internal.pixelMappingTestType;
	task.internal._HighPowerTestType			:= task.internal.highPowerTestType;

	// ========================================================================================================

	// ========================= Handle Config defaults and populate non zero zaber 2 offset postions ============
	IF Configuration.zaber2HeightArray[5] = 0 THEN
		Configuration.zaber2HeightArray[5] := 27.5; // Default
	END_IF

	IF Configuration.zaber2HeightArray[5] <> 0 THEN
		Configuration.zaber2HeightArray[0] := Configuration.zaber2HeightArray[5]- (5*Configuration.zaber2StepIndexSize_mm);
		Configuration.zaber2HeightArray[1] := Configuration.zaber2HeightArray[5]- (4*Configuration.zaber2StepIndexSize_mm);
		Configuration.zaber2HeightArray[2] := Configuration.zaber2HeightArray[5]- (3*Configuration.zaber2StepIndexSize_mm);
		Configuration.zaber2HeightArray[3] := Configuration.zaber2HeightArray[5]- (2*Configuration.zaber2StepIndexSize_mm);
		Configuration.zaber2HeightArray[4] := Configuration.zaber2HeightArray[5]- (1*Configuration.zaber2StepIndexSize_mm);

		Configuration.zaber2HeightArray[6] := Configuration.zaber2HeightArray[5]+ (1*Configuration.zaber2StepIndexSize_mm);
		Configuration.zaber2HeightArray[7] := Configuration.zaber2HeightArray[5]+ (2*Configuration.zaber2StepIndexSize_mm);
		Configuration.zaber2HeightArray[8] := Configuration.zaber2HeightArray[5]+ (3*Configuration.zaber2StepIndexSize_mm);
		Configuration.zaber2HeightArray[9] := Configuration.zaber2HeightArray[5]+ (4*Configuration.zaber2StepIndexSize_mm);
		Configuration.zaber2HeightArray[10] := Configuration.zaber2HeightArray[5]+ (5*Configuration.zaber2StepIndexSize_mm);
	END_IF

	IF Configuration.zaber2HeightCameraExpoArray[0] = 0 THEN
		Configuration.zaber2HeightCameraExpoArray[0] := 0.451; // Default
	END_IF
	IF Configuration.zaber2HeightCameraExpoArray[1] = 0 THEN
		Configuration.zaber2HeightCameraExpoArray[1] := 0.393; // Default
	END_IF
	IF Configuration.zaber2HeightCameraExpoArray[2] = 0 THEN
		Configuration.zaber2HeightCameraExpoArray[2] := 0.319; // Default
	END_IF
	IF Configuration.zaber2HeightCameraExpoArray[3] = 0 THEN
		Configuration.zaber2HeightCameraExpoArray[3] := 0.280; // Default
	END_IF
	IF Configuration.zaber2HeightCameraExpoArray[4] = 0 THEN
		Configuration.zaber2HeightCameraExpoArray[4] := 0.241; // Default
	END_IF
	IF Configuration.zaber2HeightCameraExpoArray[5] = 0 THEN
		Configuration.zaber2HeightCameraExpoArray[5] := 0.227; // Default
	END_IF
	IF Configuration.zaber2HeightCameraExpoArray[6] = 0 THEN
		Configuration.zaber2HeightCameraExpoArray[6] := 0.236; // Default
	END_IF
	IF Configuration.zaber2HeightCameraExpoArray[7] = 0 THEN
		Configuration.zaber2HeightCameraExpoArray[7] := 0.295; // Default
	END_IF
	IF Configuration.zaber2HeightCameraExpoArray[8] = 0 THEN
		Configuration.zaber2HeightCameraExpoArray[8] := 0.509; // Default
	END_IF
	IF Configuration.zaber2HeightCameraExpoArray[9] = 0 THEN
		Configuration.zaber2HeightCameraExpoArray[9] := 0.579; // Default
	END_IF
	IF Configuration.zaber2HeightCameraExpoArray[10] = 0 THEN
		Configuration.zaber2HeightCameraExpoArray[10] := 0.420; // Default
	END_IF
	// ========================================================================================================
END_ACTION
```

### Program Logical/Automation/ManualPulseLaserSFC

#### Types.typ
```iecst
TYPE
	Configuration_typ : 	STRUCT
		errorAborts : BOOL;
	END_STRUCT;
	localInterface_typ : 	STRUCT
		command : localInterfaceCommand_typ;
		status : localInterfaceStatus_typ;
		internal : localInterfaceInternal_typ;
	END_STRUCT;
	localInterfaceCommand_typ : 	STRUCT
		stop : BOOL;
		_ : BOOL;
	END_STRUCT;
	localInterfaceStatus_typ : 	STRUCT
		activeOperation : STRING[80];
		activeStep : STRING[80];
		statusMessage : STRING[vfALARMS_MAX_SNIPPET_STR_LENGTH];
		subSystemStatus : ARRAY[0..9]OF STRING[80];
		ready : BOOL;
		ErrorState : STRING[80];
		statusID : UDINT;
	END_STRUCT;
	localInterfaceInternal_typ : 	STRUCT
		PLCOpen : AtnPlcOpenStatus;
		newCommand : BOOL;
	END_STRUCT;
END_TYPE
```

#### Variables.var
```iecst
VAR
	Command : AtnPLCOpenWithParameters;
	OP_MANUAL_CALIBRATE_LASER : BOOL;
	OP_MANUAL_CALIBRATE_BEAM : BOOL;
	OP_PULSE_LASER : BOOL;
	END_TEST : BOOL;
	SKIP_PIXEL : BOOL;
	NEXT_PIXEL : BOOL;
END_VAR
```

#### commands.st
```iecst
ACTION SelectOperation:

	CASE gMachineState.operation  OF

		MACH_OP_MANUAL_CALIBRATE_LASER:
			OP_MANUAL_CALIBRATE_LASER := TRUE;
			task.status.statusID := 	ERR_FUB_BUSY;
			task.status.activeOperation:= 'Manual Pulse Laser for Laser Cal';

		MACH_OP_MANUAL_CALIBRATE_BEAM:
			OP_MANUAL_CALIBRATE_BEAM := TRUE;
			task.status.statusID := 	ERR_FUB_BUSY;
			task.status.activeOperation:= 'Manual Pulse Laser for Beam Cal';

	END_CASE

END_ACTION

ACTION ResetOperation:

	OP_MANUAL_CALIBRATE_LASER := FALSE;

END_ACTION
```

#### Cyclic.sfc
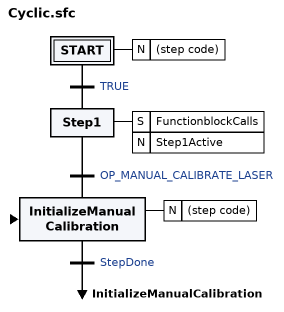
```iecst
PROGRAM _CYCLIC
INITIAL_STEP START:

SFCReset := FALSE;
END_STEP
TRANSITION FROM START TO Step1:=
TRUE
END_TRANSITION
IEC_STEP Step1:
FunctionblockCalls(S);
Step1Active(N);
END_STEP
TRANSITION FROM Step1 TO InitializeManualCalibration:=
OP_MANUAL_CALIBRATE_LASER
END_TRANSITION
STEP InitializeManualCalibration:
// initialize app with manual pulse pars
//Command.Command := gVFLCR.command.initializeManualCalibration;

//Command.Execute := TRUE;
//Command();

IF Command.Done THEN
	StepDone := TRUE;
	Command.Execute := FALSE;
	Command();
ELSE

	StepDone := FALSE;

END_IF
END_STEP
TRANSITION FROM InitializeManualCalibration TO InitializeManualCalibration:=
StepDone
END_TRANSITION
(* @SFCISJUMP := 'InitializeManualCalibration' *)
END_PROGRAM
```

#### Init.st
```iecst
PROGRAM _INIT

END_PROGRAM
```

### Program Logical/Automation/PixelMappingSFC

#### Cyclic.sfc
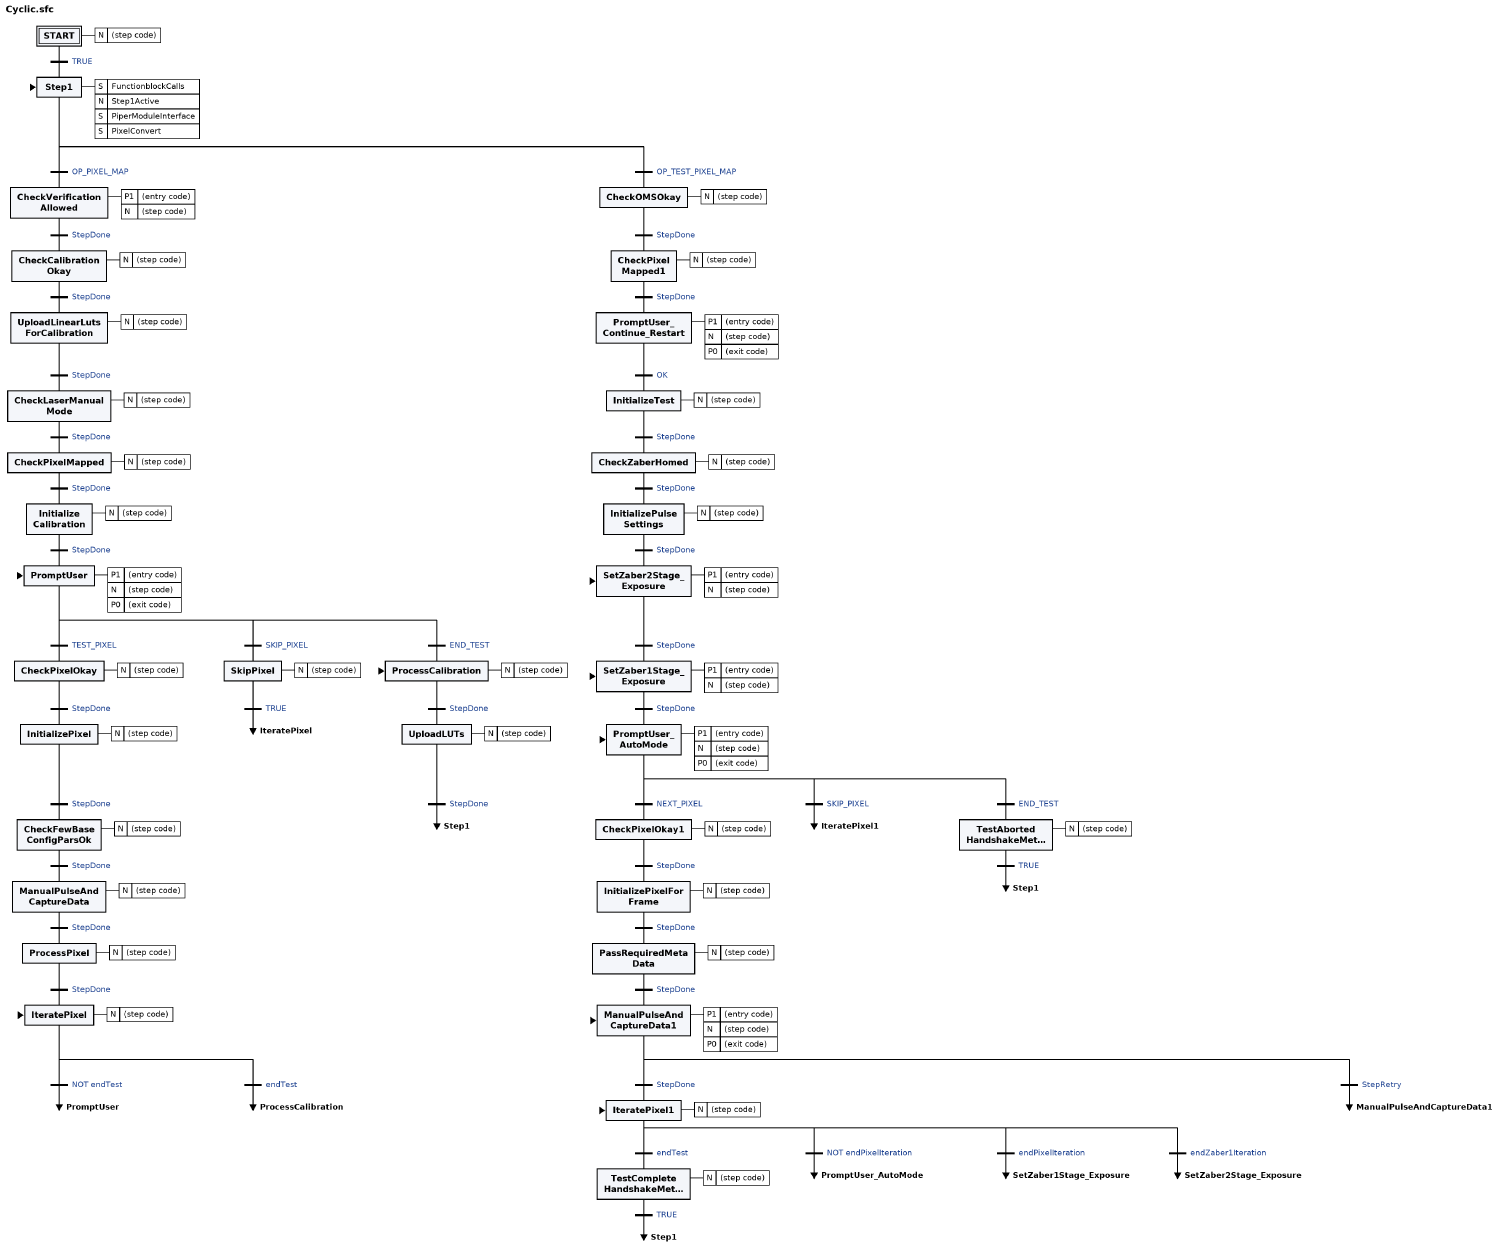
```iecst
PROGRAM _CYCLIC
INITIAL_STEP START:

SFCReset := FALSE;
END_STEP
TRANSITION FROM START TO Step1:=
TRUE
END_TRANSITION
IEC_STEP Step1:
FunctionblockCalls(S);
Step1Active(N);
PiperModuleInterface(S);
PixelConvert(S);
END_STEP
TRANSITION FROM Step1 TO CheckVerificationAllowed:=
OP_PIXEL_MAP
END_TRANSITION
TRANSITION FROM Step1 TO CheckOMSOkay:=
OP_TEST_PIXEL_MAP
END_TRANSITION
STEP CheckOMSOkay:
omsTestComplete := FALSE;
endTest := FALSE;
endPixelIteration := FALSE;

Command.Command := gVFLCR.command.checkMotionOk;
Command.Execute := TRUE;
Command();

IF Command.Done THEN
	StepDone := TRUE;
	Command.Execute := FALSE;
	Command();
ELSE
	StepDone := FALSE;
END_IF
END_STEP
TRANSITION FROM CheckOMSOkay TO CheckPixelMapped1:=
StepDone
END_TRANSITION
STEP CheckPixelMapped1:
task.status.allPixelsMapped := stateAllTrue(gVFLCR.status.pixelMapped, FALSE);

IF task.status.allPixelsMapped THEN
	StepDone := TRUE;
ELSE
	StepDone := FALSE;

	Command.Command := gVFLCR.command.laserRackRemap;

	Command.Execute := TRUE;
	Command();

	IF Command.Done THEN
		StepDone := TRUE;
		Command.Execute := FALSE;
		Command();
	ELSIF Command.Error THEN
		StepError := TRUE;
	END_IF

END_IF
END_STEP
TRANSITION FROM CheckPixelMapped1 TO PromptUser_Continue_Restart:=
StepDone
END_TRANSITION
STEP PromptUser_Continue_Restart:

IF messageHandler.msgId = 0 THEN

	CONTINUE_TEST := FALSE;
	RESTART_TEST := FALSE;

	messageHandler.msgId := MessageBox_AddMsg(ADR('Would you like to continue test or restart where you stopped last'),
	ADR('Continue'), ADR(CONTINUE_TEST),
	ADR('Restart'), ADR(RESTART_TEST));

ELSIF messageHandler.msgId <> 0 THEN

	//Waiting for the user

END_IF

IF messageHandler.cancel THEN
	messageHandler.cancel := 0;
	messageHandler.msgId := 0;
	SFCReset := TRUE;
	gMachine.IN.CMD.Stop:= TRUE;
END_IF

//Once a selection is made we are good
IF RESTART_TEST THEN

	task.internal.activeZaber1Index := 0;
	task.internal.activeZaber2Index := 0;
	task.internal.activePixelIndex := 0;

	OK := TRUE;
	MessageBox_RemoveMsg( messageHandler.msgId );
	messageHandler.msgId := 0;

ELSIF CONTINUE_TEST THEN

	OK := TRUE;
	MessageBox_RemoveMsg( messageHandler.msgId );
	messageHandler.msgId := 0;

END_IF
END_STEP
ENTRY_ACTION
messageHandler.ok := FALSE;
messageHandler.cancel := FALSE;
messageHandler.msgId := 0;
CONTINUE_TEST := FALSE;
RESTART_TEST := FALSE;
OK := FALSE;
END_ACTION
EXIT_ACTION
CONTINUE_TEST := FALSE;
RESTART_TEST := FALSE;
END_ACTION
TRANSITION FROM PromptUser_Continue_Restart TO InitializeTest:=
OK
END_TRANSITION
STEP InitializeTest:

// initialize test
// init meta writer; Zome Zaber

Command.Command := gVFLCR.command.initializeOmsTest;

Command.Execute := TRUE;
Command();

IF Command.Done THEN
	StepDone := TRUE;
	Command.Execute := FALSE;
	Command();

ELSE
	StepDone := FALSE;
END_IF
END_STEP
TRANSITION FROM InitializeTest TO CheckZaberHomed:=
StepDone
END_TRANSITION
STEP CheckZaberHomed:
Command.Command := gVFLCR.command.checkZaberHomed;

Command.Execute := TRUE;
Command();

IF Command.Done THEN
	StepDone := TRUE;
	Command.Execute := FALSE;
	Command();
ELSE
	StepDone := FALSE;
END_IF
END_STEP
TRANSITION FROM CheckZaberHomed TO InitializePulseSettings:=
StepDone
END_TRANSITION
STEP InitializePulseSettings:
// initialize app with manual pulse pars; Will create directories for calibration test as well- Should be ok; Assuming data backup of last test to Nas is done by then
Command.Command := gVFLCR.command.initializeCalibration;

Command.pParameters := ADR(gManualPulseTypeSelected);
Command.sParameters := SIZEOF(gManualPulseTypeSelected);

Command.Execute := TRUE;
Command();

IF Command.Done THEN
	StepDone := TRUE;
	Command.Execute := FALSE;
	Command();
ELSE

	StepDone := FALSE;

END_IF
END_STEP
TRANSITION FROM InitializePulseSettings TO SetZaber2Stage_Exposure:=
StepDone
END_TRANSITION
STEP SetZaber2Stage_Exposure:

// Set Zaber height and camera exposure
Command.Command := gVFLCR.command.setZaber2PosAndExposure;

Command.pParameters := ADR(task.internal.adjustZaber2AndCamera);
Command.sParameters := SIZEOF(task.internal.adjustZaber2AndCamera);

Command.Execute := TRUE;
Command();

IF Command.Done THEN
	StepDone := TRUE;
	Command.Execute := FALSE;
	Command();
ELSE

	StepDone := FALSE;

END_IF
END_STEP
ENTRY_ACTION

brsmemset( ADR(task.internal.adjustZaber2AndCamera), 0, SIZEOF(task.internal.adjustZaber2AndCamera) );

task.internal.adjustZaber2AndCamera.ZaberAbsolutePos_mm := Configuration.zaber2HeightArray[task.internal.activeZaber2Index];
task.internal.adjustZaber2AndCamera.ZaberMoveAbsolute := TRUE ;
task.internal.adjustZaber2AndCamera.CameraExposure := Configuration.zaber2HeightCameraExpoArray[task.internal.activeZaber2Index];
END_ACTION
TRANSITION FROM SetZaber2Stage_Exposure TO SetZaber1Stage_Exposure:=
StepDone
END_TRANSITION
STEP SetZaber1Stage_Exposure:

// Set Zaber height and camera exposure
Command.Command := gVFLCR.command.setZaber1PosAndExposure;

Command.pParameters := ADR(task.internal.adjustZaber1AndCamera);
Command.sParameters := SIZEOF(task.internal.adjustZaber1AndCamera);

Command.Execute := TRUE;
Command();

IF Command.Done THEN
	StepDone := TRUE;
	Command.Execute := FALSE;
	Command();
ELSE

	StepDone := FALSE;

END_IF
END_STEP
ENTRY_ACTION

brsmemset( ADR(task.internal.adjustZaber1AndCamera), 0, SIZEOF(task.internal.adjustZaber1AndCamera) );

task.internal.adjustZaber1AndCamera.ZaberAbsolutePos_mm := Configuration.zaber1HeightArray[task.internal.activeZaber1Index];
task.internal.adjustZaber1AndCamera.ZaberMoveAbsolute := TRUE ;
task.internal.adjustZaber1AndCamera.CameraExposure := Configuration.zaber1HeightCameraExpoArray[task.internal.activeZaber1Index];
END_ACTION
TRANSITION FROM SetZaber1Stage_Exposure TO PromptUser_AutoMode:=
StepDone
END_TRANSITION
STEP PromptUser_AutoMode:

IF NOT autoMode THEN
	IF messageHandler.msgId = 0 THEN

		NEXT_PIXEL := FALSE;
		SKIP_PIXEL := FALSE;
		END_TEST := FALSE;

		IF task.internal.activePixelIndex >= MACHINE_NUM_LASERS_TOTAL THEN

			// there are no more pixels
			messageHandler.msgId := MessageBox_AddMsg(ADR('There are no more pixels to test.'),
			ADR('End the test'), ADR(END_TEST),
			0, 0);

		ELSIF gVFLCR.status.vfpMap[task.internal.activePixelIndex, 1] = FALSE THEN

			// pixel is disabled
			messageHandler.msgId := MessageBox_AddMsg(ADR('Pixel is disabled. What would you like to do next?'),
			ADR('Skip pixel'), ADR(SKIP_PIXEL),
			ADR('End the test'), ADR(END_TEST));

		ELSE

			// pixel is enabled
			messageHandler.msgId := MessageBox_Add3BtnMsg(ADR('What would you like to do next?'),
			ADR('Next pixel'), ADR(NEXT_PIXEL),
			ADR('Skip pixel'), ADR(SKIP_PIXEL),
			ADR('End the test'), ADR(END_TEST));

		END_IF

	ELSIF messageHandler.msgId <> 0 THEN

		//Waiting for the user

	END_IF

	IF messageHandler.cancel THEN
		messageHandler.cancel := 0;
		messageHandler.msgId := 0;
		SFCReset := TRUE;
		gMachine.IN.CMD.Stop:= TRUE;
	END_IF

	//Once a selection is made we are good
	IF NEXT_PIXEL OR SKIP_PIXEL OR END_TEST THEN

		OK := TRUE;
		MessageBox_RemoveMsg( messageHandler.msgId );
		messageHandler.msgId := 0;

	END_IF
ELSE
	IF gVFLCR.status.vfpMap[task.internal.activePixelIndex, 1] = FALSE THEN
		SKIP_PIXEL := TRUE;
	ELSE
		NEXT_PIXEL := TRUE;
	END_IF
END_IF
END_STEP
ENTRY_ACTION
messageHandler.ok := FALSE;
messageHandler.cancel := FALSE;
messageHandler.msgId := 0;
NEXT_PIXEL := FALSE;
SKIP_PIXEL := FALSE;
END_TEST := FALSE;
OK := FALSE;
END_ACTION
EXIT_ACTION
NEXT_PIXEL := FALSE;
SKIP_PIXEL := FALSE;
END_TEST := FALSE;
END_ACTION
TRANSITION FROM PromptUser_AutoMode TO CheckPixelOkay1:=
NEXT_PIXEL
END_TRANSITION
TRANSITION FROM PromptUser_AutoMode TO IteratePixel1:=
SKIP_PIXEL
END_TRANSITION
(* @SFCISJUMP := 'IteratePixel1' *)
TRANSITION FROM PromptUser_AutoMode TO TestAbortedHandshakeMetaWriter:=
END_TEST
END_TRANSITION
STEP TestAbortedHandshakeMetaWriter:
Command.Command := gVFLCR.command.passAbortedHandshake;

Command.Execute := TRUE;
Command();

IF Command.Done THEN
	StepDone := TRUE;
	Command.Execute := FALSE;
	Command();
ELSE
	StepDone := FALSE;
END_IF
END_STEP
TRANSITION FROM TestAbortedHandshakeMetaWriter TO Step1:=
TRUE
END_TRANSITION
(* @SFCISJUMP := 'Step1' *)
STEP CheckPixelOkay1:
Command.Command := gVFLCR.command.checkMotionOk;
Command.Execute := TRUE;
Command();

IF Command.Done THEN
	StepDone := TRUE;
	Command.Execute := FALSE;
	Command();
ELSE
	StepDone := FALSE;
END_IF

END_STEP
TRANSITION FROM CheckPixelOkay1 TO InitializePixelForFrame:=
StepDone
END_TRANSITION
STEP InitializePixelForFrame:
Command.Command := gVFLCR.command.initializePixelForFrame;

task.internal.initializePixelParameters.activePixelIndex := task.internal.activePixelIndex;

Command.pParameters := ADR(task.internal.initializePixelParameters);
Command.sParameters := SIZEOF(task.internal.initializePixelParameters);

Command.Execute := TRUE;
Command();

IF Command.Done THEN
	StepDone := TRUE;
	Command.Execute := FALSE;
	Command();
ELSE

	StepDone := FALSE;

END_IF
END_STEP
TRANSITION FROM InitializePixelForFrame TO PassRequiredMetaData:=
StepDone
END_TRANSITION
STEP PassRequiredMetaData:
Command.Command := gVFLCR.command.passRequiredMetaData;

Command.Execute := TRUE;
Command();

IF Command.Done THEN
	StepDone := TRUE;
	Command.Execute := FALSE;
	Command();
ELSE
	StepDone := FALSE;
END_IF
END_STEP
TRANSITION FROM PassRequiredMetaData TO ManualPulseAndCaptureData1:=
StepDone
END_TRANSITION
STEP ManualPulseAndCaptureData1:
Command.Command := gVFLCR.command.manualPulse;

Command.pParameters := ADR(task.internal.manualPulse);
Command.sParameters := SIZEOF(task.internal.manualPulse);

Command.Execute := TRUE;
Command();

IF Command.Done THEN
	StepDone := TRUE;
	task.internal.failedImageCaptureRetry := 0;
	Command.Execute := FALSE;
	Command();
ELSIF Command.Error THEN
	IF task.internal.failedImageCaptureRetry < task.internal.numOfRetries THEN
		StepRetry := TRUE;
		task.internal.failedImageCaptureRetry := task.internal.failedImageCaptureRetry +1;
		Command.Execute := FALSE;
		Command();
	ELSE
		task.internal.failedImageCaptureRetry := 0;
		StepDone := FALSE;
		StepRetry := FALSE;
		StepError := TRUE;
		Command.Execute := FALSE;
		Command();
	END_IF
ELSE
	StepDone := FALSE;
END_IF
END_STEP
ENTRY_ACTION
task.internal.numOfRetries := 3;
END_ACTION
EXIT_ACTION
StepRetry := FALSE;
END_ACTION
TRANSITION FROM ManualPulseAndCaptureData1 TO IteratePixel1:=
StepDone
END_TRANSITION
TRANSITION FROM ManualPulseAndCaptureData1 TO ManualPulseAndCaptureData1:=
StepRetry
END_TRANSITION
(* @SFCISJUMP := 'ManualPulseAndCaptureData1' *)
STEP IteratePixel1:
task.internal.activePixelIndex := task.internal.activePixelIndex + 1;

IF task.internal.activePixelIndex >= MACHINE_NUM_LASERS_TOTAL THEN
	IF task.internal.activeZaber1Index < 10 AND task.internal.activeZaber2Index < 10 THEN // 0-10 point reading with 5 being zero offset position and 5 reading on either side
		// reset pixel iterator
		task.internal.activePixelIndex := 0;
		endPixelIteration := TRUE;
		task.internal.activeZaber1Index := task.internal.activeZaber1Index + 1;
		task.internal.currentZaber1Height := task.internal.activeZaber1Index - 1;
		endTest := FALSE;
	ELSIF task.internal.activeZaber1Index >= 10 AND task.internal.activeZaber2Index < 10 THEN
		task.internal.activePixelIndex := 0;
		endZaber1Iteration := TRUE;
		task.internal.activeZaber2Index := task.internal.activeZaber2Index + 1;
		task.internal.currentZaber2Height := task.internal.activeZaber2Index - 1;
		task.internal.activeZaber1Index := 0;
		endTest := FALSE;
	ELSE
		endTest := TRUE;
	END_IF
ELSE
	endPixelIteration := FALSE;
	endZaber1Iteration := FALSE;
	endTest := FALSE;
END_IF
END_STEP
TRANSITION FROM IteratePixel1 TO TestCompleteHandshakeMetaWriter:=
endTest
END_TRANSITION
TRANSITION FROM IteratePixel1 TO PromptUser_AutoMode:=
NOT endPixelIteration
END_TRANSITION
(* @SFCISJUMP := 'PromptUser_AutoMode' *)
TRANSITION FROM IteratePixel1 TO SetZaber1Stage_Exposure:=
endPixelIteration
END_TRANSITION
(* @SFCISJUMP := 'SetZaber1Stage_Exposure' *)
TRANSITION FROM IteratePixel1 TO SetZaber2Stage_Exposure:=
endZaber1Iteration
END_TRANSITION
(* @SFCISJUMP := 'SetZaber2Stage_Exposure' *)
STEP TestCompleteHandshakeMetaWriter:
endTest := FALSE;

Command.Command := gVFLCR.command.passCompleteHandshake;

Command.Execute := TRUE;
Command();

IF Command.Done THEN
	StepDone := TRUE;
	omsTestComplete := TRUE;
	Command.Execute := FALSE;
	Command();
ELSE
	StepDone := FALSE;
END_IF
END_STEP
TRANSITION FROM TestCompleteHandshakeMetaWriter TO Step1:=
TRUE
END_TRANSITION
(* @SFCISJUMP := 'Step1' *)
STEP CheckVerificationAllowed:
IF (task.internal.dirtyVerificationTestType OR
	task.internal.lowPowerTestType OR
	task.internal.cleanVerificationTestType) AND
	(gVFLCR.status.calibrationLUT[0] = 99999 OR
	gVFLCR.status.calibrationLUT[1] = 99999 OR
	gVFLCR.status.calibrationLUT[2] = 99999 OR
	gVFLCR.status.calibrationLUT[3] = 99999) THEN

	StepError := TRUE;
ELSE
	StepDone := TRUE;
END_IF

END_STEP
ENTRY_ACTION
StepError := FALSE;
StepDone := FALSE;
END_ACTION
TRANSITION FROM CheckVerificationAllowed TO CheckCalibrationOkay:=
StepDone
END_TRANSITION
STEP CheckCalibrationOkay:
Command.Command := gVFLCR.command.checkMotionOk;
Command.Execute := TRUE;
Command();

IF Command.Done THEN
	StepDone := TRUE;
	Command.Execute := FALSE;
	Command();
ELSE
	StepDone := FALSE;
END_IF

END_STEP
TRANSITION FROM CheckCalibrationOkay TO UploadLinearLutsForCalibration:=
StepDone
END_TRANSITION
STEP UploadLinearLutsForCalibration:
IF gManualPulseTypeSelected = VFLCR_TEST_TYPE_CALIBRATION THEN
	Command.Command := gVFLCR.command.uploadLUTs;

	task.internal.uploadLUTParameters.Calibrated := FALSE;

	Command.pParameters := ADR(task.internal.uploadLUTParameters);
	Command.sParameters := SIZEOF(task.internal.uploadLUTParameters);

	Command.Execute := TRUE;
	Command();

	IF Command.Done THEN
		StepDone := TRUE;
		Command.Execute := FALSE;
		Command();
	ELSE

		StepDone := FALSE;

	END_IF
ELSE
	StepDone := TRUE;
END_IF
END_STEP
TRANSITION FROM UploadLinearLutsForCalibration TO CheckLaserManualMode:=
StepDone
END_TRANSITION
STEP CheckLaserManualMode:
IF stateAllTrue(gVFLCR.status.manualModeEnabled,FALSE) THEN
	StepDone := TRUE;
ELSE
	StepDone := FALSE;

	Command.Command := gVFLCR.command.enableManualMode;

	Command.Execute := TRUE;
	Command();

	IF Command.Done THEN
		StepDone := TRUE;
		Command.Execute := FALSE;
		Command();
	ELSIF Command.Error THEN
		StepError := TRUE;
	END_IF

END_IF

END_STEP
TRANSITION FROM CheckLaserManualMode TO CheckPixelMapped:=
StepDone
END_TRANSITION
STEP CheckPixelMapped:
task.status.allPixelsMapped := stateAllTrue(gVFLCR.status.pixelMapped, FALSE);

IF task.status.allPixelsMapped THEN
	StepDone := TRUE;
ELSE
	StepDone := FALSE;

	Command.Command := gVFLCR.command.laserRackRemap;

	Command.Execute := TRUE;
	Command();

	IF Command.Done THEN
		StepDone := TRUE;
		Command.Execute := FALSE;
		Command();
	ELSIF Command.Error THEN
		StepError := TRUE;
	END_IF

END_IF
END_STEP
TRANSITION FROM CheckPixelMapped TO InitializeCalibration:=
StepDone
END_TRANSITION
STEP InitializeCalibration:
// reset pixel iterator
task.internal.activePixelIndex := 0;

// initialize app with manual pulse pars
Command.Command := gVFLCR.command.initializeCalibration;

Command.pParameters := ADR(gManualPulseTypeSelected);
Command.sParameters := SIZEOF(gManualPulseTypeSelected);

Command.Execute := TRUE;
Command();

IF Command.Done THEN
	StepDone := TRUE;
	Command.Execute := FALSE;
	Command();
ELSE

	StepDone := FALSE;

END_IF
END_STEP
TRANSITION FROM InitializeCalibration TO PromptUser:=
StepDone
END_TRANSITION
STEP PromptUser:
IF NOT autoMode THEN
	IF messageHandler.msgId = 0 THEN

		TEST_PIXEL := FALSE;
		SKIP_PIXEL := FALSE;
		END_TEST := FALSE;

		IF task.internal.activePixelIndex >= MACHINE_NUM_LASERS_TOTAL THEN

			// there are no more pixels
			messageHandler.msgId := MessageBox_AddMsg(ADR('There are no more pixels to test.'),
			ADR('End the test'), ADR(END_TEST),
			0, 0);

		ELSIF gVFLCR.status.vfpMap[task.internal.activePixelIndex, 1] = FALSE THEN

			// pixel is disabled
			messageHandler.msgId := MessageBox_AddMsg(ADR('Pixel is disabled. What would you like to do next?'),
			ADR('Skip pixel'), ADR(SKIP_PIXEL),
			ADR('End the test'), ADR(END_TEST));

		ELSE

			// pixel is enabled
			messageHandler.msgId := MessageBox_Add3BtnMsg(ADR('What would you like to do next?'),
			ADR('Test pixel'), ADR(TEST_PIXEL),
			ADR('Skip pixel'), ADR(SKIP_PIXEL),
			ADR('End the test'), ADR(END_TEST));

		END_IF

	ELSIF messageHandler.msgId <> 0 THEN

		//Waiting for the user

	END_IF

	IF messageHandler.cancel THEN
		messageHandler.cancel := 0;
		messageHandler.msgId := 0;
		SFCReset := TRUE;
		gMachine.IN.CMD.Stop:= TRUE;
	END_IF

	//Once a selection is made we are good
	IF TEST_PIXEL OR SKIP_PIXEL OR END_TEST THEN

		OK := TRUE;
		MessageBox_RemoveMsg( messageHandler.msgId );
		messageHandler.msgId := 0;

	END_IF
ELSE
	IF gVFLCR.status.vfpMap[task.internal.activePixelIndex, 1] = FALSE THEN
		SKIP_PIXEL := TRUE;
	ELSE
		TEST_PIXEL := TRUE;
	END_IF
END_IF
END_STEP
ENTRY_ACTION
messageHandler.ok := FALSE;
messageHandler.cancel := FALSE;
messageHandler.msgId := 0;
TEST_PIXEL := FALSE;
SKIP_PIXEL := FALSE;
END_TEST := FALSE;
OK := FALSE;
END_ACTION
EXIT_ACTION
TEST_PIXEL := FALSE;
SKIP_PIXEL := FALSE;
END_TEST := FALSE;
END_ACTION
TRANSITION FROM PromptUser TO CheckPixelOkay:=
TEST_PIXEL
END_TRANSITION
TRANSITION FROM PromptUser TO SkipPixel:=
SKIP_PIXEL
END_TRANSITION
STEP SkipPixel:
//continue
END_STEP
TRANSITION FROM SkipPixel TO IteratePixel:=
TRUE
END_TRANSITION
(* @SFCISJUMP := 'IteratePixel' *)
TRANSITION FROM PromptUser TO ProcessCalibration:=
END_TEST
END_TRANSITION
STEP ProcessCalibration:
Command.Command := gVFLCR.command.processCalibration;

Command.pParameters := 0;
Command.sParameters := 0;

Command.Execute := TRUE;
Command();

IF Command.Done THEN
	StepDone := TRUE;
	Command.Execute := FALSE;
	Command();
ELSE

	StepDone := FALSE;

END_IF
END_STEP
TRANSITION FROM ProcessCalibration TO UploadLUTs:=
StepDone
END_TRANSITION
STEP UploadLUTs:
IF gManualPulseTypeSelected = VFLCR_TEST_TYPE_CALIBRATION THEN
	Command.Command := gVFLCR.command.uploadLUTs;

	task.internal.uploadLUTParameters.Calibrated := TRUE;

	Command.pParameters := ADR(task.internal.uploadLUTParameters);
	Command.sParameters := SIZEOF(task.internal.uploadLUTParameters);

	Command.Execute := TRUE;
	Command();

	IF Command.Done THEN
		StepDone := TRUE;
		Command.Execute := FALSE;
		Command();
	ELSE

		StepDone := FALSE;

	END_IF
ELSE
	StepDone := TRUE;
END_IF
END_STEP
TRANSITION FROM UploadLUTs TO Step1:=
StepDone
END_TRANSITION
(* @SFCISJUMP := 'Step1' *)
STEP CheckPixelOkay:
Command.Command := gVFLCR.command.checkMotionOk;
Command.Execute := TRUE;
Command();

IF Command.Done THEN
	StepDone := TRUE;
	Command.Execute := FALSE;
	Command();
ELSE
	StepDone := FALSE;
END_IF

END_STEP
TRANSITION FROM CheckPixelOkay TO InitializePixel:=
StepDone
END_TRANSITION
STEP InitializePixel:
Command.Command := gVFLCR.command.initializePixel;

task.internal.initializePixelParameters.activePixelIndex := task.internal.activePixelIndex;

Command.pParameters := ADR(task.internal.initializePixelParameters);
Command.sParameters := SIZEOF(task.internal.initializePixelParameters);

Command.Execute := TRUE;
Command();

IF Command.Done THEN
	StepDone := TRUE;
	Command.Execute := FALSE;
	Command();
ELSE

	StepDone := FALSE;

END_IF
END_STEP
TRANSITION FROM InitializePixel TO CheckFewBaseConfigParsOk:=
StepDone
END_TRANSITION
STEP CheckFewBaseConfigParsOk:
//Checking few base config values are good before manual pulse
task.status.manualPulseConfigOk := stateAllTrue(gVFLCR.status.calibrationConfigParOk, FALSE);
IF task.status.manualPulseConfigOk THEN
	StepDone := TRUE;
ELSE
	//TO DO: add alarm
	StepDone := FALSE;
END_IF
END_STEP
TRANSITION FROM CheckFewBaseConfigParsOk TO ManualPulseAndCaptureData:=
StepDone
END_TRANSITION
STEP ManualPulseAndCaptureData:
Command.Command := gVFLCR.command.manualPulse;

Command.pParameters := ADR(task.internal.manualPulse);
Command.sParameters := SIZEOF(task.internal.manualPulse);

Command.Execute := TRUE;
Command();

IF Command.Done THEN
	StepDone := TRUE;
	Command.Execute := FALSE;
	Command();
ELSE

	StepDone := FALSE;

END_IF
END_STEP
TRANSITION FROM ManualPulseAndCaptureData TO ProcessPixel:=
StepDone
END_TRANSITION
STEP ProcessPixel:
Command.Command := gVFLCR.command.processPixel;

Command.pParameters := 0;
Command.sParameters := 0;

Command.Execute := TRUE;
Command();

IF Command.Done THEN
	StepDone := TRUE;
	Command.Execute := FALSE;
	Command();
ELSE

	StepDone := FALSE;

END_IF
END_STEP
TRANSITION FROM ProcessPixel TO IteratePixel:=
StepDone
END_TRANSITION
STEP IteratePixel:
task.internal.activePixelIndex := task.internal.activePixelIndex + 1;
task.internal.currentPixel := task.internal.activePixelIndex -1;

IF task.internal.activePixelIndex >= MACHINE_NUM_LASERS_TOTAL THEN
	endTest := TRUE;
ELSE
	endTest := FALSE;
END_IF
END_STEP
TRANSITION FROM IteratePixel TO PromptUser:=
NOT endTest
END_TRANSITION
(* @SFCISJUMP := 'PromptUser' *)
TRANSITION FROM IteratePixel TO ProcessCalibration:=
endTest
END_TRANSITION
(* @SFCISJUMP := 'ProcessCalibration' *)
END_PROGRAM
```

### VFLCR.typ
```iecst
TYPE
	VFLCRApi_typ : 	STRUCT
		command : VFLCRApiCommand_typ;
		status : VFLCRApiStatus_typ;
		IO : VFLCRApiIO_typ;
		alarm : VFLCRApiAlarm_typ;
	END_STRUCT;
	VFLCRApiCommand_typ : 	STRUCT
		openLayer : STRING[80];
		resetSoftwareError : STRING[80];
		abortLayer : STRING[80];
		resetAllErrors : STRING[80];
		deleteLaserControlFiles : STRING[80];
	END_STRUCT;
	VFLCRApiStatus_typ : 	STRUCT
		rackOnline : STRING[80];
		layerOpen : STRING[80];
	END_STRUCT;
	VFLCRApiIO_typ : 	STRUCT
		rack : STRING[80];
	END_STRUCT;
	VFLCRApiAlarm_typ : 	STRUCT
		components : vfAlarms_Component_typ;
		AGGREGATE_GENERAL_ALARM : vfAlarms_Instance_type;
		AGGREGATE_HARDWARE_ALARM : vfAlarms_Instance_type;
		AGGREGATE_SOFTWARE_ALARM : vfAlarms_Instance_type;
		AGGREGATE_PIXELMAPPING_ALARM : vfAlarms_Instance_type;
		AGGREGATE_CALIBAPP_ALARM : vfAlarms_Instance_type;
		VFLCR_HW_HEARTBEAT_ERROR_AL9100 : vfAlarms_Instance_type;
		VFLCR_HW_HARDWARE_ERROR_AL9103 : vfAlarms_Instance_type;
		VFLCR_HW_SUPPLY_FAN_FAIL_AL9104 : vfAlarms_Instance_type;
		VFLCR_HW_SUPPLY_OVERTEMP_AL9105 : vfAlarms_Instance_type;
		VFLCR_HW_SUPPLY_AC_LOW_AL9106 : vfAlarms_Instance_type;
		VFLCR_HW_SUPPLY_DC_FAIL_AL9107 : vfAlarms_Instance_type;
		VFLCR_HW_CONTROL_POWER_AL9108 : vfAlarms_Instance_type;
		VFLCR_HW_LASER_READY_FAIL_AL9109 : vfAlarms_Instance_type;
		VFLCR_HW_LASER_MAIN_POWER_AL9110 : vfAlarms_Instance_type;
		VFLCR_HW_LASER_EMISSION_AL9111 : vfAlarms_Instance_type;
		VFLCR_HW_LASER_FATAL_AL9112 : vfAlarms_Instance_type;
		VFLCR_HW_LASER_WATCHDOG_AL9113 : vfAlarms_Instance_type;
		VFLCR_HW_POWERLINK_ERROR_AL9114 : vfAlarms_Instance_type;
		VFLCR_SW_VERSION_MISMATCH_AL9200 : vfAlarms_Instance_type;
		VFLCR_SW_ID_MISMATCH_AL9201 : vfAlarms_Instance_type;
		VFLCR_SW_LUT_LOAD_FAIL_AL9202 : vfAlarms_Instance_type;
		VFLCR_SW_MAP_UNDEFINED_AL9203 : vfAlarms_Instance_type;
		VFLCR_SW_SYSTEM_ERROR_AL9204 : vfAlarms_Instance_type;
		VFLCR_SW_TRAJECTORY_ERROR_AL9205 : vfAlarms_Instance_type;
		VFLCR_SW_PRINT_NOT_READY_AL9206 : vfAlarms_Instance_type;
		VFLCR_SW_COMMAND_INHIBIT_AL9207 : vfAlarms_Instance_type;
		VFLCR_PM_FILE_NOT_FOUND_AL9300 : vfAlarms_Instance_type;
		VFLCR_PM_PATH_NOT_FOUND_AL9301 : vfAlarms_Instance_type;
		VFLCR_PM_FILE_OPEN_ERROR_AL9302 : vfAlarms_Instance_type;
		VFLCR_PM_FILE_CLOSE_ERROR_AL9303 : vfAlarms_Instance_type;
		VFLCR_PM_FILE_READ_ERROR_AL9304 : vfAlarms_Instance_type;
		VFLCR_PM_FILE_DATA_ERROR_AL9305 : vfAlarms_Instance_type;
		VFLCR_PM_VERSION_CONFLICT_AL9306 : vfAlarms_Instance_type;
		VFLCR_PM_IGNORED_PIXEL_AL9307 : vfAlarms_Instance_type;
		VFLCR_PM_RANGE_EXCEEDED_AL9308 : vfAlarms_Instance_type;
		VFLCR_APP_HEARTBEAT_ERROR_AL9400 : vfAlarms_Instance_type;
		VFLCR_APP_COMMAND_TIMEOUT_AL9401 : vfAlarms_Instance_type;
		VFLCR_APP_CMD_B4_READY_AL9402 : vfAlarms_Instance_type;
		VFLCR_APP_RESULTS_TIMEOUT_AL9403 : vfAlarms_Instance_type;
		VFLCR_APP_BUCKET_MISSING_AL9404 : vfAlarms_Instance_type;
		VFLCR_APP_S3_CONNECTION_AL9405 : vfAlarms_Instance_type;
		VFLCR_APP_CAPTURE_FAILED_AL9406 : vfAlarms_Instance_type;
		VFLCR_DISABLE_CHILLER_RUN_AL9208 : vfAlarms_Instance_type;
		VFLCR_DISABLE_OB_FLOW_LOW_AL9209 : vfAlarms_Instance_type;
		PIXEL_ENABLE_MISMATCH_AL9309 : vfAlarms_Instance_type;
		VFLCR_VERIFY_INHIBIT_AL9210 : vfAlarms_Instance_type;
	END_STRUCT;
	VFLCROpenLayerCommandPars_typ : 	STRUCT
		parameters : VFLCROpenLayerParameters_typ;
	END_STRUCT;
	VFLCROpenLayerRackPars_typ : 	STRUCT
		Rack : USINT;
	END_STRUCT;
	VFLCROpenLayerParameters_typ : 	STRUCT
		selectedBuildLayout : UDINT;
		selectedPrintNumber : UINT;
		selectedLayer : UDINT;
	END_STRUCT;
	LaserSnippets_typ : 	STRUCT
		rackNumber : USINT;
		laserNumber : USINT;
		pixelNumber : USINT;
		supplyNumber : USINT;
		additionalInfoLaserFatal : STRING[160];
	END_STRUCT;
END_TYPE
```

### VFLCR.var
```iecst
(*Constants defining capabilities of each VF-LCR system...*)
(*Machine-specific constants...*)
VAR CONSTANT
	MACHINE_NUM_LASER_RACKS : USINT := 4; (*Number of VF-LCR controlled laser racks*)
	MACHINE_MAI_LASER_RACKS : USINT := MACHINE_NUM_LASER_RACKS-1;
END_VAR
(*Test type constants*)
(*Rack/laser to pixel mapping and vice-versa...*)
(*Global ATN interface*)
VAR
	gVFLCR : VFLCRApi_typ;
	gLaserSnippets : LaserSnippets_typ;
END_VAR
```

### Program Logical/ProcessControl/VFLCR/VFLCR_System (IEC) - VF-LCR System Control

#### Main.st - Init, cyclic, exit code
```iecst
PROGRAM _INIT

	Name := 'LCR System';

END_PROGRAM

PROGRAM _CYCLIC

	// VF-LCR code is based on Gen 2 v3.18.0

	///////////////////////////////////////////////////////////////
	// API:
	//	Requires:
	//	- nothing
	//	Commands:
	//	- manualPulse 				- Sets up parameters and distributes the manual pulse commands to the VFLCR_Operations
	//	- manualPulseAbort 			- Cancel all manual pulse commands
	//  Statuses:
	//	- cycleOKFailCount_PLK2		- the number of cycles that had a Powerlink cycle error
	//	- syncOKFailCount_PLK2		- the number of cycles that had a Powerlink synchronization error
	//	- plkErrorDetected			- there is a Powerlink cycle or synchronization error
	//	- manualModeEnabled			- manual mode is enabled for all racks, respecting ignores
	//	- autoModeEnabled			- auto mode is enabled for all racks, respecting ignores
	//	Inhbitits:
	//	- nothing
	///////////////////////////////////////////////////////////////

	// Call Piper
	//PiperModuleInterface;

	// Read in external components

	// Read external states

	IF task.command.rebootPLC THEN
		task.internal.rebootPLC := TRUE;
	END_IF

	IF task.command.confirmReboot  THEN

		task.internal.rebootPLC := FALSE;
		SYSreset(TRUE, SYSLIB_WARMSTART);

	END_IF

	IF task.command.closePopup THEN

		task.internal.rebootPLC := FALSE;

	END_IF

	// Error reset command
	IF task.command.resetAllErrors THEN
		executeCommand(gVFLCR.command.resetAllErrors);
	END_IF

	// Layer commands
	IF task.command.openLayer THEN
		// pars set by hmi
		task.internal.openLayerCommand.Execute := TRUE;
	END_IF

	IF task.command.abortLayer THEN
		task.internal.atnSystemCommand.Command := gVFLCR.command.abortLayer;
		task.internal.atnSystemCommand.Execute := TRUE;
	END_IF

	task.internal.openLayerCommand.Command := gVFLCR.command.openLayer;
	task.internal.openLayerCommand.pParameters := ADR(task.parameters.openLayer);
	task.internal.openLayerCommand.sParameters := SIZEOF(task.parameters.openLayer);
	task.internal.openLayerCommand();
	task.internal.openLayerCommand.Execute := FALSE;

	// If we get an abort command, ensure that the manual pulse start gets errored

	task.internal.atnSystemCommand();
	task.internal.atnSystemCommand.Execute := FALSE;

	task.status.racksOnline := stateAllTrue(gVFLCR.status.rackOnline, FALSE);

END_PROGRAM

PROGRAM _EXIT

END_PROGRAM
```

#### Types.typ - Local data types
```iecst
TYPE
	localInterface_typ : 	STRUCT
		command : localInterfaceCommand_typ;
		parameters : localInterfaceParameter_typ;
		status : localInterfaceStatus_typ;
		internal : localInterfaceInternal_typ;
	END_STRUCT;
	localInterfaceCommand_typ : 	STRUCT
		openLayer : BOOL;
		resetAllErrors : BOOL;
		closePopup : BOOL;
		confirmReboot : BOOL;
		rebootPLC : BOOL;
		abortLayer : BOOL;
	END_STRUCT;
	localInterfaceParameter_typ : 	STRUCT
		openLayer : VFLCROpenLayerCommandPars_typ;
	END_STRUCT;
	POWER_SEQUENCE :
		(
		SEQUENCE_READY,
		SEQUENCE_ENABLING_DC_POWER,
		SEQUENCE_ENABLING_LASER_EMISSION,
		SEQUENCE_ENABLING_LASER_POWER,
		SEQUENCE_ENABLING_LASER_MOD,
		SEQUENCE_FAILED
		);
	localInterfaceStatus_typ : 	STRUCT
		cycleOKFailCount_PLK2 : UINT;
		syncOKFailCount_PLK2 : UINT;
		statusMessage : STRING[vfALARMS_MAX_SNIPPET_STR_LENGTH];
		racksOnline : BOOL;
	END_STRUCT;
	LaserManualPulseCalculated_typ : 	STRUCT
		pixelNumber : UINT;
		startingPowerWatts : REAL;
		powerIncrementWatts : REAL;
		endingPowerWatts : REAL;
		endingPowerHigh : REAL;
	END_STRUCT;
	localInterfaceInternal_typ : 	STRUCT
		atnSystemCommand : AtnPLCOpen;
		enableLaserPowerSequenceCommand : AtnPLCOpen;
		openLayerCommand : AtnPLCOpenWithParameters;
		rebootPLC : BOOL;
		PLCOpen : AtnPlcOpenStatus;
	END_STRUCT;
	IO_typ : 	STRUCT
		di : IODI_typ;
	END_STRUCT;
	IODI_typ : 	STRUCT
		cycleOK_PLK2 : BOOL;
		syncOK_PLK2 : BOOL;
	END_STRUCT;
	vflcrSystemCommandStatus_typ : 	STRUCT
		enableDCPower : commandStatus_typ;
		enableLaserPower : commandStatus_typ;
		enableLaserEmission : commandStatus_typ;
		enableLaserFullSequence : commandStatus_typ;
	END_STRUCT;
	commandStatus_typ : 	STRUCT
		busy : BOOL;
		idle : BOOL;
	END_STRUCT;
END_TYPE
```

#### Variables.var - Local variables
```iecst
VAR
	Name : STRING[80];
	IO : IO_typ;
	task : localInterface_typ;
	index : INT;
	active : BOOL;
	FoundActive : BOOL;
	moduleName : STRING[256];
	i : USINT;
END_VAR
```

#### PiperInterface.st
```iecst
(********************************************************************
 * COPYRIGHT --
 ********************************************************************
 * Program: MachineProg
 * File: PiperModuleInterface.st
 * Author: Josh
 * Created: October 03, 2013
 ********************************************************************
 * Implementation of program MachineProg
 ********************************************************************)

ACTION PiperModuleInterface:

	// Give this module a name so it is easier to debug
	ModuleInterface.ModuleName:= Name;

	// Add a module to the Piper
	Module.ModuleInterface:= ADR(ModuleInterface);
	Module.Piper:= ADR(gMachine);
	Module();

	// Set machine mode optional actions
	piperEnableLasers := FALSE;
	CASE gMachineModeApi.status.activeMode OF

		MACHINE_MODE_MAINTENANCE:

		MACHINE_MODE_SETUP:

		MACHINE_MODE_PRODUCTION:

			//only reset the lasers if its good to do so..
			IF stateAllTrue(gMachineModeApi.watchdog.productionModeOkay, FALSE) THEN
				piperEnableLasers := TRUE;
			END_IF

		ELSE

	END_CASE

	// Handle any machine states that this module needs to respond to
	CASE ModuleInterface.PiperState OF
//		MACH_ST_BOOTING:
//		MACH_ST_CLEARING:
//		MACH_ST_STOPPED:
//		MACH_ST_STARTING:
//		MACH_ST_IDLE:
//		MACH_ST_SUSPENDED:
//		MACH_ST_EXECUTE:
		MACH_ST_STOPPING:

			IF _prevPiperState <> ModuleInterface.PiperState THEN

				executeCommand(gVFLCR.command.abortLayer);
				executeCommand(gVFLCR.command.manualPulseAbort);
			END_IF

			ModuleInterface.ModuleResponse := ModuleInterface.PiperState;

		MACH_ST_ABORTING:

			piperCommands.disableDCPower := TRUE;

			CASE ModuleInterface.PiperSubState OF
				SUB_STATE_INIT:
					ModuleInterface.ModuleSubStateRequest := SUB_STATE_DEPOWER_LASERS;

				SUB_STATE_DEPOWER_LASERS:

					IF stateAllFalse(gVFLCR.status.dcPowerEnabled, TRUE) THEN
						IF _prevPiperState <> ModuleInterface.PiperState THEN
							executeCommand(gVFLCR.command.abortLayer);
						END_IF

						ModuleInterface.ModuleResponse := ModuleInterface.PiperState;
					END_IF

			END_CASE

//		MACH_ST_ABORTED:
//		MACH_ST_HOLDING:
//		MACH_ST_HELD:
//		MACH_ST_UNHOLDING:
//		MACH_ST_SUSPENDING:
//		MACH_ST_UNSUSPENDING:
			//		MACH_ST_STARTING,

		MACH_ST_RESETTING:

			IF piperEnableLasers AND stateAnyFalse(gVFLCR.status.readyToPrint, FALSE) THEN

				piperCommands.resetAllErrors := TRUE;

				CASE ModuleInterface.PiperSubState OF
					SUB_STATE_INIT:
						ModuleInterface.ModuleSubStateRequest := SUB_STATE_CONFIRM_LASERS_WANTED;

					SUB_STATE_CONFIRM_LASERS_WANTED:

						IF (messageHandler.msgId = 0) AND NOT(ModuleInterface.ModuleSubStateRequest = SUB_STATE_RESETTING_LASERS_ON) THEN
							messageHandler.msgId := MessageBox_AddMsg(ADR('Turn on Lasers?'),
							ADR('Yes'), ADR(messageHandler.ok),
							ADR('No'), ADR(messageHandler.cancel));
						END_IF

						IF messageHandler.ok THEN
							ModuleInterface.ModuleSubStateRequest := SUB_STATE_RESETTING_LASERS_ON;
							messageHandler.ok := FALSE;
							messageHandler.msgId := 0;
						END_IF

						IF messageHandler.cancel THEN
							ModuleInterface.ModuleResponse := ModuleInterface.PiperState;
							messageHandler.cancel := FALSE;
							messageHandler.msgId := 0;
						END_IF

					SUB_STATE_RESETTING_LASERS_ON:

						piperCommands.enableAllLaserFunctions := TRUE;

						IF stateAllTrue(gVFLCR.status.readyToPrint, FALSE) OR gSimulation THEN
							ModuleInterface.ModuleResponse := ModuleInterface.PiperState;
						END_IF

				END_CASE

			ELSE

				ModuleInterface.ModuleResponse := ModuleInterface.PiperState;

			END_IF

//		MACH_ST_COMPLETING:
//		MACH_ST_COMPLETE:

		MACH_ST_BYPASSED:

		ELSE
			ModuleInterface.ModuleResponse:= ModuleInterface.PiperState;

	END_CASE

	// Turn level commands to edges
	EdgePosArray(ADR(piperCommands), ADR(_piperCommands), ADR(task.command), SIZEOF(task.command));
	brsmemset(ADR(piperCommands), 0, SIZEOF(piperCommands));

	_prevPiperState := ModuleInterface.PiperState;
END_ACTION
```

#### PiperModule.var - Local variables
```iecst
(********************************************************************
 * COPYRIGHT --
 ********************************************************************
 * Program: PiperModuleTemplate
 * File: PiperModuleTemplate.var
 * Author: Josh
 * Created: October 03, 2013
 ********************************************************************
 * Local variables of program PiperModuleTemplate
 ********************************************************************)
VAR
	ModuleInterface : Module_Interface_typ;
	Module : Piper_Module_Fub;
	piperCommands : localInterfaceCommand_typ;
	_piperCommands : localInterfaceCommand_typ;
	piperEnableLasers : BOOL;
	messageHandler : MessageHandler_typ;
	_prevPiperState : MACH_ST_enum;
END_VAR
```

#### hmiHelper.st
```iecst
ACTION hmiHelper:

	//for the loader icon to tell if the sequence is running or not
	task.internal.hmiCommandStatus.enableLaserFullSequence.busy := task.internal.hmiCommandStatus.enableDCPower.busy OR task.internal.hmiCommandStatus.enableLaserEmission.busy OR task.internal.hmiCommandStatus.enableLaserPower.busy;
	task.internal.hmiCommandStatus.enableLaserFullSequence.idle := NOT(task.internal.hmiCommandStatus.enableLaserFullSequence.busy);

	//DC power
	IF (brsstrcmp(ADR(task.internal.atnSystemCommand.Command),ADR(gVFLCR.command.enableDCPower))=0) THEN
		task.internal.hmiCommandStatus.enableDCPower.busy := task.internal.atnSystemCommand.Busy;
	ELSE
		task.internal.hmiCommandStatus.enableDCPower.busy := FALSE;
	END_IF
	task.internal.hmiCommandStatus.enableDCPower.idle := NOT(task.internal.hmiCommandStatus.enableDCPower.busy);

	//laser emission
	IF (brsstrcmp(ADR(task.internal.atnSystemCommand.Command),ADR(gVFLCR.command.enableLaserEmission))=0) THEN
		task.internal.hmiCommandStatus.enableLaserEmission.busy := task.internal.atnSystemCommand.Busy;
	ELSE
		task.internal.hmiCommandStatus.enableLaserEmission.busy := FALSE;
	END_IF
	task.internal.hmiCommandStatus.enableLaserEmission.idle := NOT(task.internal.hmiCommandStatus.enableLaserEmission.busy);

	//laser power
	IF (brsstrcmp(ADR(task.internal.atnSystemCommand.Command),ADR(gVFLCR.command.enableLaserPower))=0) THEN
		task.internal.hmiCommandStatus.enableLaserPower.busy := task.internal.atnSystemCommand.Busy;
	ELSE
		task.internal.hmiCommandStatus.enableLaserPower.busy := FALSE;
	END_IF
	task.internal.hmiCommandStatus.enableLaserPower.idle := NOT(task.internal.hmiCommandStatus.enableLaserPower.busy);

END_ACTION
```

### Program Logical/ProcessControl/VFLCR/VFLCR_Operation (IEC) - VF-LCR Operations

#### Main.st - Init, cyclic, exit code
```iecst
PROGRAM _INIT

	//brsitoa(Configuration.rackIndex + 1, ADR(moduleName));
	moduleName := CONCAT('VF-LCR Rack ', moduleName);

	subscribePLCOpenWithParameters(gVFLCR.command.openLayer, moduleName, ADR(task.internal.openLayerCommandParameters), SIZEOF(task.internal.openLayerCommandParameters),task.command.openLayer, task.internal.PLCOpenOpenLayer);
	subscribePLCOpen(gVFLCR.command.abortLayer, moduleName, task.command.abortLayer, task.internal.PLCOpenAbortLayer);

	subscribePLCOpen(gVFLCR.command.deleteLaserControlFiles, moduleName, task.command.deleteLaserControlFiles, task.internal.PLCOpenDeleteLaserControlFiles);

	registerStateBool(gVFLCR.status.rackOnline, moduleName, task.status.commsOK);

	task.internal.abortLayerTON.PT := T#5s;
	task.internal.deleteLaserControlFilesTON.PT := T#5s;
	task.internal.openLayerTON.PT := T#5s;

	subscribeCommandBool(gVFLCR.command.resetAllErrors, moduleName, task.command.resetSoftwareError);

END_PROGRAM

PROGRAM _CYCLIC
	///////////////////////////////////////////////////////////////

	//	- openLayer 				- Opens a layer
	//	- abortLayer 				- Aborts a layer

	//	- deleteLaserControlFiles 	- Deletes laser control files from the VF-LCR system

	// Read in external components
	ReadInputIO;

	IF gSimulation THEN
		SimulateIO;
	END_IF

	// Read external states
	task.status.ready := TRUE;

	///////////////////////////////////////////////////////////////
	// Handle interpreting commands that do not require STATE_READY
	///////////////////////////////////////////////////////////////
	IF task.status.ready THEN

		IF task.command.deleteLaserControlFiles THEN
			task.internal.newCommand := TRUE;
		END_IF

	ELSE // Not ready

		task.status.state := STATE_NOT_READY;

	END_IF

	///////////////////////////////////////////////////////////////
	// Handle any canceled commands that are required
	///////////////////////////////////////////////////////////////

		IF task.command.abortLayer THEN

			IO.do.AbortLayer := TRUE;

		END_IF

		IF IO.di.LayerAborted THEN

			IO.do.AbortLayer := FALSE;
			task.internal.PLCOpenAbortLayer.status := ERR_OK;

		ELSIF task.internal.abortLayerTON.Q THEN

			IO.do.AbortLayer := FALSE;
			task.internal.PLCOpenAbortLayer.status := VFLCR_ERROR;

		END_IF

		IF task.command.resetSoftwareError THEN

			IO.do.ClearLaserErrors := TRUE;

		END_IF

		IF task.command.deleteLaserControlFiles THEN

			IO.do.Delete_LaserControlFiles := TRUE;

		END_IF

		IF IO.di.LaserControlFiles_Deleted THEN

			IO.do.Delete_LaserControlFiles := FALSE;
			task.internal.PLCOpenDeleteLaserControlFiles.status := ERR_OK;

		ELSIF task.internal.deleteLaserControlFilesTON.Q THEN

			IO.do.Delete_LaserControlFiles := FALSE;
			task.internal.PLCOpenDeleteLaserControlFiles.status := VFLCR_ERROR;

		END_IF

		IF task.command.openLayer THEN

			IF task.internal.PLCOpenOpenLayer.parametersWritten THEN
				task.parameters.openLayerParameters := task.internal.openLayerCommandParameters.parameters;

				IF  (task.parameters.openLayerParameters.selectedPrintNumber > 0) AND NOT (IO.di.LayerOpen) THEN
					IO.do.OpenLayer := TRUE;
				ELSE
					IO.do.OpenLayer := FALSE;
					task.internal.PLCOpenOpenLayer.status := VFLCR_ERROR;
				END_IF
			ELSE
				// we need pars
				task.internal.PLCOpenOpenLayer.status := VFLCR_ERROR;
			END_IF

		END_IF

		IF IO.di.LayerOpen THEN

			// Unlike other commands, IO.do.OpenLayer must stay set after a success (while the layer is open)
			task.internal.PLCOpenOpenLayer.status := ERR_OK;

		ELSIF task.internal.openLayerTON.Q THEN

			// Timeout cancels the command, so lower IO
			IO.do.OpenLayer := FALSE;
			task.internal.PLCOpenOpenLayer.status := VFLCR_ERROR;

		END_IF

		// Check for layer not being open
		// EDGEPOS must be first so its internal fub always runs
		IF EDGEPOS(IO.di.LayerClosed OR IO.di.LayerAborted OR IO.di.LayerError OR task.command.abortLayer) THEN

			IO.do.OpenLayer := FALSE;
			task.internal.PLCOpenOpenLayer.status := VFLCR_ERROR;

		END_IF

	// Reset statuses/internals that aren't checked every cycle
	task.status.commsOK := TRUE;
	task.status.commsError := FALSE;

	task.internal.abortLayerTON.IN := IO.do.AbortLayer AND NOT IO.di.LayerAborted;
	task.internal.abortLayerTON();

	task.internal.deleteLaserControlFilesTON.IN := IO.do.Delete_LaserControlFiles AND NOT IO.di.LaserControlFiles_Deleted;
	task.internal.deleteLaserControlFilesTON();

	task.internal.openLayerTON.IN := IO.do.OpenLayer AND NOT IO.di.LayerOpen;
	task.internal.openLayerTON();

	///////////////////////////////////////////////////////////////
	// Reset all commands to ensure they don't get buffered
	///////////////////////////////////////////////////////////////
	brsmemset(ADR(task.command), 0, SIZEOF(task.command));

	task.internal.newCommand := FALSE;

	// Handle output IO
	WriteOutputIO;

END_PROGRAM

PROGRAM _EXIT

	// On program exit, disable all lasers, force current layer to be aborted, and disable both AUTO and MANUAL modes.
	ShutDownIO;

END_PROGRAM
```

#### Types.typ - Local data types
```iecst
TYPE
	Configuration_typ : 	STRUCT
		rackIndex : USINT;
	END_STRUCT;
	LaserOperation_typ : 	STRUCT
		command : LaserOperationCommand_typ;
		parameters : LaserOperationParameter_typ;
		status : LaserOperationStatus_typ;
		internal : LaserOperationInternal_typ;
	END_STRUCT;
	LaserOperationCommand_typ : 	STRUCT
		openLayer : BOOL;
		resetSoftwareError : BOOL;
		abortLayer : BOOL;
		deleteLaserControlFiles : BOOL;
	END_STRUCT;
	LaserOperationParameter_typ : 	STRUCT
		openLayerParameters : VFLCROpenLayerParameters_typ;
	END_STRUCT;
	LaserOperationStatus_typ : 	STRUCT
		ready : BOOL;
		state : STATE;
		sequence : SEQUENCE;
		commsOK : BOOL;
		commsError : BOOL;
		layerOpen : BOOL;
	END_STRUCT;
	LaserOperationInternal_typ : 	STRUCT
		localLockout : BOOL;
		newCommand : BOOL;
		previousState : STATE;
		PLCOpenAbortLayer : AtnPlcOpenStatus;
		PLCOpenDeleteLaserControlFiles : AtnPlcOpenStatus;
		PLCOpenOpenLayer : AtnPlcOpenStatus;
		abortLayerTON : TON;
		resetSoftwareErrorTON : TON;
		deleteLaserControlFilesTON : TON;
		openLayerCommandParameters : VFLCROpenLayerCommandPars_typ;
		openLayerTON : TON;
	END_STRUCT;
	LaserOperationAlarmID_typ : 	STRUCT
		AL9100 : UDINT;
		AL9104 : UDINT;
		AL9105 : UDINT;
		AL9106 : UDINT;
		AL9107 : UDINT;
		AL9109 : UDINT;
		AL9110 : UDINT;
		AL9111 : UDINT;
		AL9112 : UDINT;
		AL9113 : UDINT;
		AL9202 : UDINT;
	END_STRUCT;
	STATE :
		(
		STATE_NOT_READY,
		STATE_READY
		);
	SEQUENCE :
		(
		SEQUENCE_IDLE,
		SEQUENCE_ERROR,
		SEQUENCE_DONE
		);
	LaserIO_typ : 	STRUCT
		di : LaserIODI_typ;
		do : LaserIODO_typ;
		ai : LaserIOAI_typ;
		ao : LaserIOAO_typ;
		raw : LaserIORaw_typ; (*IO that gets converted to/from meaningful vars above.*)
	END_STRUCT;
	LaserIORaw_typ : 	STRUCT
		iFPGARevision : UDINT;
		iSoftwareRevision : UDINT;
		iSystemStatus : UDINT;
		iOperationStatus : UDINT;
		iLaserReady_Error : UDINT;
		iLaserControlPowerEnabled : UDINT;
		iLaserMainPowerEnabled : UDINT;
		iLaserEmissionEnabled : UDINT;
		iLaserFatalError : UDINT;
		iLaserWatchdogError : UDINT;
		iManualModeLaserPower : UDINT;
		oSystemControl : UDINT;
		oOperationControl : UDINT;
		oLaserEnable : UDINT;
		oEnableLaserMainPower : UDINT;
		oEnableGuideLaser : UDINT;
		oEnableLaserEmission : UDINT;
		oResetLaserErrors : UDINT;
		oManualLaserCurrentSetpoint : UDINT;
		oIndirectRegisterRequestAddress : UDINT; (*target address for write to VFLCR*)
		oIndirectRegisterRequestData : UDINT; (*data from target address for write to VFLCR*)
		iIndirectRegisterResponseAddress : UDINT; (*read the requested address from VFLCR*)
		iIndirectRegisterResponseData : UDINT; (*read the data from the requested address from VFLCR*)
		oManualLaserOperation : UDINT;
	END_STRUCT;
	LaserIODI_typ : 	STRUCT
		PoweLinkModuleOK : BOOL;
		LaserControlFiles_Deleted : BOOL;
		LayerOpen : BOOL;
		LayerAborted : BOOL;
		LayerClosed : BOOL;
		LayerError : BOOL;
	END_STRUCT;
	LaserIODO_typ : 	STRUCT
		Delete_LaserControlFiles : BOOL; (*OperationControl.1*)
		Transfer_LaserControlFiles : BOOL; (*OperationControl.3*)
		EnableMode_MANUAL : BOOL; (*OperationControl.8*)
		OpenLayer : BOOL; (*OperationControl.8*)
		ClearLaserErrors : BOOL; (*OperationControl.9*)
		AbortLayer : BOOL; (*OperationControl.9*)
	END_STRUCT;
	LaserIOAI_typ : 	STRUCT
		SystemHeartbeat : UDINT; (*Heartbeat from the VF-LCR*)
		FPGAVersion : UINT;
		FPGARevision : UINT;
		SoftwareVersion : UINT;
		SoftwareRevision : UINT;
		LUTFiles_CalibrationID : UDINT;
		SelectedLaser_DMAStatus : UDINT;
		SelectedLaser_DMATrajectory : UDINT;
		SelectedLaser_DMALastPacket : UDINT;
	END_STRUCT;
	LaserIOAO_typ : 	STRUCT
		PLCHeartbeat : UDINT;
		SelectedBuildLayout : UDINT;
		SelectedPrintNumber : UDINT;
		SelectedLayerNumber : UDINT;
		StartingTrajectoryNumber : UDINT;
	END_STRUCT;
END_TYPE
```

#### Variables.var - Local variables
```iecst
VAR RETAIN
	Configuration : Configuration_typ;
END_VAR
VAR
	task : LaserOperation_typ;
	currentSupply : USINT;
	currentLaser : USINT;
	index : USINT;
	rackIndex : USINT;
	laserIndex : USINT;
	pixelIndex : USINT;
	bitIndex : USINT;
	scanMicrosec : UDINT;
	allLasersDisabled : BOOL;
	moduleName : STRING[80];
	IO : LaserIO_typ;
	RTInfo_0 : RTInfo;
	pixelEnableMismatch : STRING[80];
	i : UDINT;
	ii : UDINT;
END_VAR
```

#### Powerlink.st
```iecst
ACTION ReadInputIO:

		IO.ai.FPGAVersion :=  UDINT_TO_UINT(SHR(IO.raw.iFPGARevision, 16));
		IO.ai.FPGARevision := UDINT_TO_UINT(IO.raw.iFPGARevision AND 16#FFFF);

		IO.ai.SoftwareVersion :=  UDINT_TO_UINT(SHR(IO.raw.iSoftwareRevision, 16));
		IO.ai.SoftwareRevision := UDINT_TO_UINT(IO.raw.iSoftwareRevision AND 16#FFFF);

		// -----------------
		// Operation Status
		// -----------------
		//IO.di.LUTFiles_Deleted := BIT_TST(IO.raw.iOperationStatus, 0);
		IO.di.LaserControlFiles_Deleted := BIT_TST(IO.raw.iOperationStatus, 1);
		//IO.di.LUTFiles_LoadSuccess := BIT_TST(IO.raw.iOperationStatus, 2);
		//IO.di.LUTFiles_LoadFailure := BIT_TST(IO.raw.iOperationStatus, 3);

		//IO.di.ModeEnabled_MANUAL := BIT_TST(IO.raw.iOperationStatus, 6);
		//IO.di.ModeEnabled_AUTO := BIT_TST(IO.raw.iOperationStatus, 7);
		IO.di.LayerOpen := BIT_TST(IO.raw.iOperationStatus, 8);
		IO.di.LayerAborted := BIT_TST(IO.raw.iOperationStatus, 9);
		IO.di.LayerClosed := BIT_TST(IO.raw.iOperationStatus, 10);
		IO.di.LayerError := BIT_TST(IO.raw.iOperationStatus, 11);

		//IO.di.SystemWatchdogFailure := BIT_TST(IO.raw.iOperationStatus, 14);
		//IO.di.SystemOperational := BIT_TST(IO.raw.iOperationStatus, 15);

		// Simulation
		IF gSimulation THEN
			SimulateIO;
		END_IF

END_ACTION

ACTION WriteOutputIO:

		// -----------------
		// Heartbeats
		// -----------------
		// Continuously increment heartbeat to VF-LCR system.
		IO.ao.PLCHeartbeat := IO.ao.PLCHeartbeat + 1;

		// -----------------
		// Layer Selection
		// -----------------
		IO.ao.SelectedBuildLayout := task.parameters.openLayerParameters.selectedBuildLayout;
		IO.ao.SelectedPrintNumber := task.parameters.openLayerParameters.selectedPrintNumber;
		IO.ao.SelectedLayerNumber := task.parameters.openLayerParameters.selectedLayer;

		// -----------------
		// Operation Control
		// -----------------
		//IF (IO.do.Delete_LUTFiles) THEN
		//	IO.raw.oOperationControl := BIT_SET(IO.raw.oOperationControl, 0);
		//ELSE
		//	IO.raw.oOperationControl := BIT_CLR(IO.raw.oOperationControl, 0);
		//END_IF

		IF (IO.do.Delete_LaserControlFiles) THEN
			IO.raw.oOperationControl := BIT_SET(IO.raw.oOperationControl, 1);
		ELSE
			IO.raw.oOperationControl := BIT_CLR(IO.raw.oOperationControl, 1);
		END_IF

		//IF (IO.do.Transfer_LUTFiles) THEN
		//	IO.raw.oOperationControl := BIT_SET(IO.raw.oOperationControl, 2);
		//ELSE
		//	IO.raw.oOperationControl := BIT_CLR(IO.raw.oOperationControl, 2);
	//END_IF

		IF (IO.do.ClearLaserErrors) THEN
			IO.raw.oOperationControl := BIT_SET(IO.raw.oOperationControl, 13);
		ELSE
			IO.raw.oOperationControl := BIT_CLR(IO.raw.oOperationControl, 13);
		END_IF

		IF (IO.do.Transfer_LaserControlFiles) THEN
			IO.raw.oOperationControl := BIT_SET(IO.raw.oOperationControl, 3);
		ELSE
			IO.raw.oOperationControl := BIT_CLR(IO.raw.oOperationControl, 3);
		END_IF

		IF (IO.do.EnableMode_MANUAL) THEN
			IO.raw.oOperationControl := BIT_SET(IO.raw.oOperationControl, 6); // Set manual mode
			IO.raw.oOperationControl := BIT_CLR(IO.raw.oOperationControl, 7); // Clear auto mode
		ELSE
			IO.raw.oOperationControl := BIT_CLR(IO.raw.oOperationControl, 6); // Clear manual mode
			IO.raw.oOperationControl := BIT_SET(IO.raw.oOperationControl, 7); // Set auto mode
		END_IF

		IF (IO.do.OpenLayer) THEN
			IO.raw.oOperationControl := BIT_SET(IO.raw.oOperationControl, 8);
		ELSE
			IO.raw.oOperationControl := BIT_CLR(IO.raw.oOperationControl, 8);
		END_IF

		IF (IO.do.AbortLayer) THEN
			IO.raw.oOperationControl := BIT_SET(IO.raw.oOperationControl, 9);
		ELSE
			IO.raw.oOperationControl := BIT_CLR(IO.raw.oOperationControl, 9);
		END_IF

		FOR index := 0 TO 21 DO
			IO.raw.oLaserEnable := BIT_SET(IO.raw.oLaserEnable, index);
		END_FOR

END_ACTION

ACTION ShutDownIO:

	IO.raw.oEnableLaserMainPower := 0;
	IO.raw.oEnableLaserEmission := 0;
	IO.raw.oManualLaserOperation := 0;
	IO.raw.oOperationControl := BIT_CLR(IO.raw.oOperationControl, 6); // Disable MANUAL mode
	IO.raw.oOperationControl := BIT_CLR(IO.raw.oOperationControl, 7); // Disable AUTO mode
	IO.raw.oOperationControl := BIT_SET(IO.raw.oOperationControl, 9); // Force AbortLayer command

END_ACTION
```

#### Simulation.st
```iecst
ACTION SimulateIO:

	IO.di.LaserControlFiles_Deleted := IO.do.Delete_LaserControlFiles;

	IO.di.LayerAborted := IO.do.AbortLayer;
	IO.di.LayerOpen	:= IO.do.OpenLayer;

END_ACTION
```

#### SubSequence.st - not listed in the package file held
```iecst
ACTION EnableSuppliesSubSequence:

	CASE task.status.sequence OF

SEQUENCE_ENABLE_DC_POWER_START:

			// Enable power supply IO with a 1.5s delay between each
			IF currentSupply < VFLCR_NUM_POWER_SUPPLIES THEN

				IO.do.LaserPowerSupply[currentSupply] := NOT(Configuration.ignoreSupply[currentSupply]);
				task.internal.delayTON.PT := T#1500ms;
				task.internal.delayTON.IN := TRUE;

				IF task.internal.delayTON.Q THEN

					task.internal.delayTON.IN := FALSE; // Handles resetting before the next supply and before the laser check
					currentSupply := currentSupply + 1;

				END_IF

			ELSE

				task.status.sequence := SEQUENCE_ENABLE_DC_POWER_CHECK;

			END_IF

		SEQUENCE_ENABLE_DC_POWER_CHECK:

			// Wait 20s for laser system check
			task.internal.delayTON.PT := T#5s;
			task.internal.delayTON.IN := TRUE;

			IF task.internal.delayTON.Q THEN

				task.internal.delayTON.IN := FALSE;
				task.status.dcPowerEnabled := TRUE;
				task.status.sequence := SEQUENCE_DONE;

			END_IF

	END_CASE

END_ACTION

ACTION EnableLasersSubSequence:

	CASE task.status.sequence OF

		SEQUENCE_ENABLE_LASERS_START:

			// Enable laser power IO with a 250ms delay between each
			IF currentLaser < VFLCR_NUM_LASERS THEN

				IO.do.EnableLaserPower[currentLaser] := NOT(Configuration.ignoreLaser[currentLaser]);
				IO.do.EnableGuideLaser[currentLaser] := FALSE; // Disable guide laser while power is on
				task.internal.delayTON.PT := T#250ms;
				task.internal.delayTON.IN := TRUE;

				IF task.internal.delayTON.Q THEN

					task.internal.delayTON.IN := FALSE; // Handles resetting before the next supply and before the status delay
					currentLaser := currentLaser + 1;

				END_IF

			ELSE

				task.status.coolingRequired := TRUE;
				task.status.sequence := SEQUENCE_ENABLE_LASERS_STATUS;

			END_IF

		SEQUENCE_ENABLE_LASERS_STATUS:

			// Wait 3.5s
			task.internal.delayTON.PT := T#3500ms;
			task.internal.delayTON.IN := TRUE;

			IF task.internal.delayTON.Q THEN

				task.internal.delayTON.IN := FALSE;
				task.status.laserPowerEnabled := TRUE;
				task.status.sequence := SEQUENCE_DONE;

			END_IF

	END_CASE

END_ACTION

ACTION ManualPulseSubSequence:

	CASE task.status.sequence OF

		SEQUENCE_MANUAL_PULSE_TRIGGER:

			task.internal.triggerFrameDataCollection.Execute := TRUE;

			//task.command.disableLaserEmission := TRUE;

			task.status.sequence := SEQUENCE_MANUAL_PULSE_RESPONSE;

		SEQUENCE_MANUAL_PULSE_RESPONSE:
			// Pixel Test
			IF stateAnyTrue( gVFLCR.status.usingGen3LaserCalibrationApp , TRUE ) AND stateAllFalse(gSFCControlApi.status.sOMSModeActive,FALSE) THEN

				// capture data after last pulse of this power level

				IF task.internal.triggerDataCollection.Done THEN

					task.status.sequence := SEQUENCE_MANUAL_PULSE_INCREMENT;

				ELSIF task.internal.triggerDataCollection.Error THEN

					task.status.sequence := SEQUENCE_ERROR;

				ELSIF NOT task.internal.triggerDataCollection.Busy THEN

					// this command forwards pulse parameters + more via plcOpen params
					task.internal.dataCollectionParameters.CurrentPowerWatts := task.status.manualPulseStatus.currentPower_W;
					task.internal.dataCollectionParameters.LaserParameters := task.parameters.manualPulseParameters;
					task.internal.triggerDataCollection.Execute := TRUE;

				END_IF
				// sOMS test
			ELSIF stateAnyTrue( gVFLCR.status.usingGen3LaserCalibrationApp , TRUE ) AND stateAnyTrue(gSFCControlApi.status.sOMSModeActive,FALSE) THEN

				// capture data after last pulse of this power level

				gOpcData_ToGen3CalibApp.LaserPulseComplete := TRUE;

				IF task.internal.triggerFrameDataCollection.Done THEN

					gOpcData_ToGen3CalibApp.LaserPulseComplete := FALSE;
					task.internal.triggerFrameDataCollection.Execute := FALSE;
					task.status.sequence := SEQUENCE_MANUAL_PULSE_INCREMENT;

				ELSIF task.internal.triggerFrameDataCollection.Error THEN

					gOpcData_ToGen3CalibApp.LaserPulseComplete := FALSE;
					task.internal.triggerFrameDataCollection.Execute := FALSE;
					task.status.sequence := SEQUENCE_ERROR;

				END_IF

			ELSE

				task.status.sequence := SEQUENCE_MANUAL_PULSE_INCREMENT;

			END_IF

		SEQUENCE_MANUAL_PULSE_INCREMENT:

			task.status.manualPulseStatus.currentStep := task.status.manualPulseStatus.currentStep + 1;

			// Check for completion
			IF task.status.manualPulseStatus.currentStep >= task.internal.parameters.manualPulseParameters.numPowerLevels THEN

				task.status.manualPulseActive := FALSE;

				task.status.sequence := SEQUENCE_DONE;

			ELSE

				task.status.sequence := SEQUENCE_MANUAL_PULSE_TRIGGER;

			END_IF

	END_CASE

END_ACTION
```

### Program Logical/ProcessControl/VFLCR/Gen3PythonLaserCalibration
